LIN {X 0,Y 467.676,Z 280.243,A -85,B 0,C 180,E1 -7671.63,E2 -7671.63} C_VEL
LIN {X 0,Y 467.961,Z 272.023,A -85,B 0,C 180,E1 -7674.393,E2 -7674.393} C_VEL
LIN {X 0,Y 468.313,Z 262.63,A -85,B 0,C 180,E1 -7677.724,E2 -7677.724} C_VEL
LIN {X 0,Y 468.659,Z 254.669,A -85,B 0,C 180,E1 -7680.654,E2 -7680.654} C_VEL
LIN {X 0,Y 469.091,Z 246.823,A -85,B 0,C 180,E1 -7683.665,E2 -7683.665} C_VEL
LIN {X 0,Y 469.381,Z 240.972,A -85,B 0,C 180,E1 -7686.046,E2 -7686.046} C_VEL
LIN {X 0,Y 468.758,Z 236.725,A -85,B 0,C 180,E1 -7687.93,E2 -7687.93} C_VEL
LIN {X 0,Y 467.6,Z 230.243,A -85,B 0,C 180,E1 -7691.113,E2 -7691.113} C_VEL
LIN {X 0,Y 467.556,Z 230.247,A -85,B 0,C 180,E1 -7693.82,E2 -7693.82} C_VEL
LIN {X 0,Y 467.557,Z 230.246,A -85,B 0,C 180,E1 -7696.255,E2 -7696.255} C_VEL
LIN {X 0,Y 467.586,Z 230.243,A -85,B 0,C 180,E1 -7698.721,E2 -7698.721} C_VEL
LIN {X 0,Y 467.577,Z 230.244,A -85,B 0,C 180,E1 -7701.406,E2 -7701.406} C_VEL
LIN {X 0,Y 467.56,Z 230.247,A -85,B 0,C 180,E1 -7704.26,E2 -7704.26} C_VEL
LIN {X 0,Y 467.582,Z 230.244,A -85,B 0,C 180,E1 -7707.32,E2 -7707.32} C_VEL
LIN {X 0,Y 467.57,Z 230.243,A -85,B 0,C 180,E1 -7710.666,E2 -7710.666} C_VEL
LIN {X 0,Y 467.628,Z 230.239,A -85,B 0,C 180,E1 -7713.199,E2 -7713.199} C_VEL
LIN {X 0,Y 467.592,Z 230.242,A -85,B 0,C 180,E1 -7716.467,E2 -7716.467} C_VEL
LIN {X 0,Y 467.623,Z 230.236,A -85,B 0,C 180,E1 -7719.776,E2 -7719.776} C_VEL
LIN {X 0,Y 467.608,Z 230.238,A -85,B 0,C 180,E1 -7722.505,E2 -7722.505} C_VEL
LIN {X 0,Y 467.604,Z 230.24,A -85,B 0,C 180,E1 -7725.195,E2 -7725.195} C_VEL
LIN {X 0,Y 467.653,Z 230.236,A -85,B 0,C 180,E1 -7727.853,E2 -7727.853} C_VEL
LIN {X 0,Y 467.679,Z 230.229,A -85,B 0,C 180,E1 -7731.356,E2 -7731.356} C_VEL
LIN {X 0,Y 467.741,Z 230.222,A -85,B 0,C 180,E1 -7733.961,E2 -7733.961} C_VEL
LIN {X 0,Y 467.857,Z 230.208,A -85,B 0,C 180,E1 -7737.416,E2 -7737.416} C_VEL
LIN {X 0,Y 467.878,Z 230.206,A -85,B 0,C 180,E1 -7739.999,E2 -7739.999} C_VEL
LIN {X 0,Y 467.855,Z 230.209,A -85,B 0,C 180,E1 -7742.581,E2 -7742.581} C_VEL
LIN {X 0,Y 467.738,Z 230.224,A -85,B 0,C 180,E1 -7746.036,E2 -7746.036} C_VEL
LIN {X 0,Y 467.676,Z 230.233,A -85,B 0,C 180,E1 -7748.641,E2 -7748.641} C_VEL
LIN {X 0,Y 467.592,Z 230.245,A -85,B 0,C 180,E1 -7751.266,E2 -7751.266} C_VEL
LIN {X 0,Y 467.277,Z 230.507,A -85,B 0,C 180,E1 -7753.923,E2 -7753.923} C_VEL
LIN {X 0,Y 467.233,Z 233.257,A -85,B 0,C 180,E1 -7756.604,E2 -7756.604} C_VEL
LIN {X 0,Y 467.155,Z 236.019,A -85,B 0,C 180,E1 -7759.326,E2 -7759.326} C_VEL
LIN {X 0,Y 467.074,Z 238.94,A -85,B 0,C 180,E1 -7762.095,E2 -7762.095} C_VEL
LIN {X 0,Y 467.043,Z 241.899,A -85,B 0,C 180,E1 -7764.917,E2 -7764.917} C_VEL
LIN {X 0,Y 466.93,Z 244.936,A -85,B 0,C 180,E1 -7767.812,E2 -7767.812} C_VEL
LIN {X 0,Y 466.869,Z 248.241,A -85,B 0,C 180,E1 -7770.903,E2 -7770.903} C_VEL
LIN {X 0,Y 466.884,Z 249.126,A -85,B 0,C 180,E1 -7771.731,E2 -7771.731} C_VEL
LIN {X 0,Y 470.12,Z 262.455,A -85,B 0,C 180,E1 -7772.256,E2 -7772.256} C_VEL
LIN {X 0,Y 470.316,Z 267.493,A -85,B 0,C 180,E1 -7772.469,E2 -7772.469} C_VEL
LIN {X 0,Y 469.881,Z 280.326,A -85,B 0,C 180,E1 -7773.115,E2 -7773.115} C_VEL
LIN {X 0,Y 469.378,Z 291.965,A -85,B 0,C 180,E1 -7773.898,E2 -7773.898} C_VEL
LIN {X 0,Y 468.916,Z 303.063,A -85,B 0,C 180,E1 -7774.846,E2 -7774.846} C_VEL
LIN {X 0,Y 468.446,Z 312.887,A -85,B 0,C 180,E1 -7775.891,E2 -7775.891} C_VEL
LIN {X 0,Y 468.022,Z 321.872,A -85,B 0,C 180,E1 -7777.077,E2 -7777.077} C_VEL
LIN {X 0,Y 467.606,Z 329.48,A -85,B 0,C 180,E1 -7778.311,E2 -7778.311} C_VEL
LIN {X 0,Y 467.302,Z 335.582,A -85,B 0,C 180,E1 -7779.53,E2 -7779.53} C_VEL
LIN {X 0,Y 467.087,Z 340.512,A -85,B 0,C 180,E1 -7780.753,E2 -7780.753} C_VEL
LIN {X 0,Y 466.944,Z 344.398,A -85,B 0,C 180,E1 -7781.972,E2 -7781.972} C_VEL
LIN {X 0,Y 466.825,Z 347.337,A -85,B 0,C 180,E1 -7783.177,E2 -7783.177} C_VEL
LIN {X 0,Y 466.665,Z 350.158,A -85,B 0,C 180,E1 -7784.943,E2 -7784.943} C_VEL
LIN {X 0,Y 466.633,Z 351.147,A -85,B 0,C 180,E1 -7786.294,E2 -7786.294} C_VEL
LIN {X 0,Y 466.618,Z 351.185,A -85,B 0,C 180,E1 -7787.56,E2 -7787.56} C_VEL
LIN {X 0,Y 466.646,Z 350.357,A -85,B 0,C 180,E1 -7788.851,E2 -7788.851} C_VEL
LIN {X 0,Y 466.745,Z 348.596,A -85,B 0,C 180,E1 -7790.165,E2 -7790.165} C_VEL
LIN {X 0,Y 466.885,Z 344.834,A -85,B 0,C 180,E1 -7791.891,E2 -7791.891} C_VEL
LIN {X 0,Y 467.095,Z 339.496,A -85,B 0,C 180,E1 -7793.536,E2 -7793.536} C_VEL
LIN {X 0,Y 467.374,Z 333.457,A -85,B 0,C 180,E1 -7794.944,E2 -7794.944} C_VEL
LIN {X 0,Y 467.669,Z 326.553,A -85,B 0,C 180,E1 -7796.219,E2 -7796.219} C_VEL
LIN {X 0,Y 468.159,Z 317.583,A -85,B 0,C 180,E1 -7797.543,E2 -7797.543} C_VEL
LIN {X 0,Y 468.545,Z 309,A -85,B 0,C 180,E1 -7798.576,E2 -7798.576} C_VEL
LIN {X 0,Y 469.032,Z 298.415,A -85,B 0,C 180,E1 -7799.614,E2 -7799.614} C_VEL
LIN {X 0,Y 469.515,Z 286.668,A -85,B 0,C 180,E1 -7800.522,E2 -7800.522} C_VEL
LIN {X 0,Y 469.957,Z 274.999,A -85,B 0,C 180,E1 -7801.227,E2 -7801.227} C_VEL
LIN {X 0,Y 470.132,Z 262.702,A -85,B 0,C 180,E1 -7801.787,E2 -7801.787} C_VEL
LIN {X 0,Y 467.551,Z 251.251,A -85,B 0,C 180,E1 -7802.245,E2 -7802.245} C_VEL
LIN {X 0,Y 466.704,Z 249.393,A -85,B 0,C 180,E1 -7802.401,E2 -7802.401} C_VEL
LIN {X 0,Y 465.362,Z 248.01,A -85,B 0,C 180,E1 -7802.739,E2 -7802.739} C_VEL
LIN {X 0,Y 462.544,Z 247.044,A -85,B 0,C 180,E1 -7803.723,E2 -7803.723} C_VEL
LIN {X 0,Y 460.557,Z 246.182,A -85,B 0,C 180,E1 -7804.819,E2 -7804.819} C_VEL
LIN {X 0,Y 459.773,Z 244.848,A -85,B 0,C 180,E1 -7805.933,E2 -7805.933} C_VEL
LIN {X 0,Y 459.817,Z 241.701,A -85,B 0,C 180,E1 -7808.797,E2 -7808.797} C_VEL
LIN {X 0,Y 459.935,Z 238.951,A -85,B 0,C 180,E1 -7811.324,E2 -7811.324} C_VEL
LIN {X 0,Y 459.981,Z 235.075,A -85,B 0,C 180,E1 -7814.946,E2 -7814.946} C_VEL
LIN {X 0,Y 460.104,Z 231.233,A -85,B 0,C 180,E1 -7818.547,E2 -7818.547} C_VEL
LIN {X 0,Y 460.424,Z 231.136,A -85,B 0,C 180,E1 -7821.22,E2 -7821.22} C_VEL
LIN {X 0,Y 460.693,Z 231.1,A -85,B 0,C 180,E1 -7823.87,E2 -7823.87} C_VEL
LIN {X 0,Y 460.81,Z 231.087,A -85,B 0,C 180,E1 -7827.378,E2 -7827.378} C_VEL
LIN {X 0,Y 460.837,Z 231.081,A -85,B 0,C 180,E1 -7830,E2 -7830} C_VEL
LIN {X 0,Y 460.81,Z 231.085,A -85,B 0,C 180,E1 -7832.623,E2 -7832.623} C_VEL
LIN {X 0,Y 460.698,Z 231.098,A -85,B 0,C 180,E1 -7836.131,E2 -7836.131} C_VEL
LIN {X 0,Y 460.614,Z 231.11,A -85,B 0,C 180,E1 -7838.777,E2 -7838.777} C_VEL
LIN {X 0,Y 460.618,Z 231.109,A -85,B 0,C 180,E1 -7842.458,E2 -7842.458} C_VEL
LIN {X 0,Y 460.584,Z 231.113,A -85,B 0,C 180,E1 -7845.999,E2 -7845.999} C_VEL
LIN {X 0,Y 460.556,Z 231.118,A -85,B 0,C 180,E1 -7848.903,E2 -7848.903} C_VEL
LIN {X 0,Y 460.55,Z 231.118,A -85,B 0,C 180,E1 -7851.484,E2 -7851.484} C_VEL
LIN {X 0,Y 460.535,Z 231.119,A -85,B 0,C 180,E1 -7854.333,E2 -7854.333} C_VEL
LIN {X 0,Y 460.57,Z 231.115,A -85,B 0,C 180,E1 -7857.244,E2 -7857.244} C_VEL
LIN {X 0,Y 460.498,Z 231.124,A -85,B 0,C 180,E1 -7860.241,E2 -7860.241} C_VEL
LIN {X 0,Y 460.517,Z 231.121,A -85,B 0,C 180,E1 -7863.326,E2 -7863.326} C_VEL
LIN {X 0,Y 460.468,Z 231.13,A -85,B 0,C 180,E1 -7866.531,E2 -7866.531} C_VEL
LIN {X 0,Y 460.568,Z 231.115,A -85,B 0,C 180,E1 -7869.859,E2 -7869.859} C_VEL
LIN {X 0,Y 460.532,Z 231.12,A -85,B 0,C 180,E1 -7872.906,E2 -7872.906} C_VEL
LIN {X 0,Y 460.515,Z 231.122,A -85,B 0,C 180,E1 -7875.83,E2 -7875.83} C_VEL
LIN {X 0,Y 460.535,Z 231.12,A -85,B 0,C 180,E1 -7878.992,E2 -7878.992} C_VEL
LIN {X 0,Y 460.539,Z 231.118,A -85,B 0,C 180,E1 -7881.271,E2 -7881.271} C_VEL
LIN {X 0,Y 460.506,Z 231.124,A -85,B 0,C 180,E1 -7884.556,E2 -7884.556} C_VEL
LIN {X 0,Y 460.527,Z 231.12,A -85,B 0,C 180,E1 -7887.718,E2 -7887.718} C_VEL
LIN {X 0,Y 460.543,Z 231.119,A -85,B 0,C 180,E1 -7890.771,E2 -7890.771} C_VEL
LIN {X 0,Y 460.559,Z 231.117,A -85,B 0,C 180,E1 -7893.737,E2 -7893.737} C_VEL
LIN {X 0,Y 460.543,Z 231.119,A -85,B 0,C 180,E1 -7896.626,E2 -7896.626} C_VEL
LIN {X 0,Y 460.549,Z 231.117,A -85,B 0,C 180,E1 -7899.455,E2 -7899.455} C_VEL
LIN {X 0,Y 460.559,Z 231.118,A -85,B 0,C 180,E1 -7902.232,E2 -7902.232} C_VEL
LIN {X 0,Y 460.564,Z 231.114,A -85,B 0,C 180,E1 -7904.967,E2 -7904.967} C_VEL
LIN {X 0,Y 460.61,Z 231.11,A -85,B 0,C 180,E1 -7908.561,E2 -7908.561} C_VEL
LIN {X 0,Y 460.619,Z 231.108,A -85,B 0,C 180,E1 -7911.225,E2 -7911.225} C_VEL
LIN {X 0,Y 460.708,Z 231.1,A -85,B 0,C 180,E1 -7913.872,E2 -7913.872} C_VEL
LIN {X 0,Y 460.801,Z 231.087,A -85,B 0,C 180,E1 -7917.379,E2 -7917.379} C_VEL
LIN {X 0,Y 460.855,Z 231.082,A -85,B 0,C 180,E1 -7920.001,E2 -7920.001} C_VEL
LIN {X 0,Y 460.801,Z 231.086,A -85,B 0,C 180,E1 -7922.624,E2 -7922.624} C_VEL
LIN {X 0,Y 460.689,Z 231.1,A -85,B 0,C 180,E1 -7926.132,E2 -7926.132} C_VEL
LIN {X 0,Y 460.623,Z 231.108,A -85,B 0,C 180,E1 -7928.778,E2 -7928.778} C_VEL
LIN {X 0,Y 460.618,Z 231.107,A -85,B 0,C 180,E1 -7932.446,E2 -7932.446} C_VEL
LIN {X 0,Y 460.605,Z 231.111,A -85,B 0,C 180,E1 -7935.999,E2 -7935.999} C_VEL
LIN {X 0,Y 460.576,Z 231.114,A -85,B 0,C 180,E1 -7938.903,E2 -7938.903} C_VEL
LIN {X 0,Y 460.521,Z 231.124,A -85,B 0,C 180,E1 -7941.487,E2 -7941.487} C_VEL
LIN {X 0,Y 460.527,Z 231.119,A -85,B 0,C 180,E1 -7944.334,E2 -7944.334} C_VEL
LIN {X 0,Y 460.564,Z 231.118,A -85,B 0,C 180,E1 -7947.246,E2 -7947.246} C_VEL
LIN {X 0,Y 460.516,Z 231.121,A -85,B 0,C 180,E1 -7950.241,E2 -7950.241} C_VEL
LIN {X 0,Y 460.526,Z 231.124,A -85,B 0,C 180,E1 -7953.326,E2 -7953.326} C_VEL
LIN {X 0,Y 460.482,Z 231.125,A -85,B 0,C 180,E1 -7956.53,E2 -7956.53} C_VEL
LIN {X 0,Y 460.533,Z 231.119,A -85,B 0,C 180,E1 -7959.863,E2 -7959.863} C_VEL
LIN {X 0,Y 460.518,Z 231.121,A -85,B 0,C 180,E1 -7962.901,E2 -7962.901} C_VEL
LIN {X 0,Y 460.513,Z 231.121,A -85,B 0,C 180,E1 -7965.831,E2 -7965.831} C_VEL
LIN {X 0,Y 460.572,Z 231.225,A -85,B 0,C 180,E1 -7968.772,E2 -7968.772} C_VEL
LIN {X 0,Y 461.795,Z 237.98,A -85,B 0,C 180,E1 -7971.885,E2 -7971.885} C_VEL
LIN {X 0,Y 462.378,Z 242.064,A -85,B 0,C 180,E1 -7973.668,E2 -7973.668} C_VEL
LIN {X 0,Y 462.268,Z 247.187,A -85,B 0,C 180,E1 -7975.769,E2 -7975.769} C_VEL
LIN {X 0,Y 461.823,Z 255.013,A -85,B 0,C 180,E1 -7978.841,E2 -7978.841} C_VEL
LIN {X 0,Y 461.394,Z 263.555,A -85,B 0,C 180,E1 -7982.064,E2 -7982.064} C_VEL
LIN {X 0,Y 460.978,Z 272.095,A -85,B 0,C 180,E1 -7985.212,E2 -7985.212} C_VEL
LIN {X 0,Y 460.666,Z 281.728,A -85,B 0,C 180,E1 -7988.534,E2 -7988.534} C_VEL
LIN {X 0,Y 460.372,Z 291.269,A -85,B 0,C 180,E1 -7991.762,E2 -7991.762} C_VEL
LIN {X 0,Y 460.171,Z 299.065,A -85,B 0,C 180,E1 -7994.352,E2 -7994.352} C_VEL
LIN {X 0,Y 462.488,Z 312.664,A -85,B 0,C 180,E1 -7994.786,E2 -7994.786} C_VEL
LIN {X 0,Y 463.263,Z 319.162,A -85,B 0,C 180,E1 -7995.054,E2 -7995.054} C_VEL
LIN {X 0,Y 462.85,Z 330.828,A -85,B 0,C 180,E1 -7995.602,E2 -7995.602} C_VEL
LIN {X 0,Y 462.346,Z 341.575,A -85,B 0,C 180,E1 -7996.26,E2 -7996.26} C_VEL
LIN {X 0,Y 461.85,Z 353.16,A -85,B 0,C 180,E1 -7997.161,E2 -7997.161} C_VEL
LIN {X 0,Y 461.377,Z 363.168,A -85,B 0,C 180,E1 -7998.133,E2 -7998.133} C_VEL
LIN {X 0,Y 460.819,Z 372.383,A -85,B 0,C 180,E1 -7999.232,E2 -7999.232} C_VEL
LIN {X 0,Y 460.42,Z 381.376,A -85,B 0,C 180,E1 -8000.555,E2 -8000.555} C_VEL
LIN {X 0,Y 460.057,Z 388.614,A -85,B 0,C 180,E1 -8001.876,E2 -8001.876} C_VEL
LIN {X 0,Y 459.851,Z 393.504,A -85,B 0,C 180,E1 -8002.977,E2 -8002.977} C_VEL
LIN {X 0,Y 459.755,Z 398.263,A -85,B 0,C 180,E1 -8004.297,E2 -8004.297} C_VEL
LIN {X 0,Y 459.581,Z 401.894,A -85,B 0,C 180,E1 -8005.614,E2 -8005.614} C_VEL
LIN {X 0,Y 459.592,Z 403.772,A -85,B 0,C 180,E1 -8006.493,E2 -8006.493} C_VEL
LIN {X 0,Y 459.572,Z 405.175,A -85,B 0,C 180,E1 -8007.37,E2 -8007.37} C_VEL
LIN {X 0,Y 459.496,Z 406.778,A -85,B 0,C 180,E1 -8009.123,E2 -8009.123} C_VEL
LIN {X 0,Y 459.475,Z 406.994,A -85,B 0,C 180,E1 -8010,E2 -8010} C_VEL
LIN {X 0,Y 459.496,Z 406.779,A -85,B 0,C 180,E1 -8010.876,E2 -8010.876} C_VEL
LIN {X 0,Y 459.572,Z 405.179,A -85,B 0,C 180,E1 -8012.629,E2 -8012.629} C_VEL
LIN {X 0,Y 459.592,Z 403.778,A -85,B 0,C 180,E1 -8013.506,E2 -8013.506} C_VEL
LIN {X 0,Y 459.635,Z 400.819,A -85,B 0,C 180,E1 -8014.824,E2 -8014.824} C_VEL
LIN {X 0,Y 459.759,Z 396.815,A -85,B 0,C 180,E1 -8016.142,E2 -8016.142} C_VEL
LIN {X 0,Y 459.928,Z 390.656,A -85,B 0,C 180,E1 -8017.683,E2 -8017.683} C_VEL
LIN {X 0,Y 460.288,Z 383.936,A -85,B 0,C 180,E1 -8019.003,E2 -8019.003} C_VEL
LIN {X 0,Y 460.701,Z 375.598,A -85,B 0,C 180,E1 -8020.325,E2 -8020.325} C_VEL
LIN {X 0,Y 461.152,Z 367.056,A -85,B 0,C 180,E1 -8021.427,E2 -8021.427} C_VEL
LIN {X 0,Y 461.674,Z 356.888,A -85,B 0,C 180,E1 -8022.492,E2 -8022.492} C_VEL
LIN {X 0,Y 462.091,Z 346.077,A -85,B 0,C 180,E1 -8023.411,E2 -8023.411} C_VEL
LIN {X 0,Y 462.652,Z 334.667,A -85,B 0,C 180,E1 -8024.178,E2 -8024.178} C_VEL
LIN {X 0,Y 463.12,Z 322.971,A -85,B 0,C 180,E1 -8024.781,E2 -8024.781} C_VEL
LIN {X 0,Y 462.988,Z 316.237,A -85,B 0,C 180,E1 -8025.063,E2 -8025.063} C_VEL
LIN {X 0,Y 460.789,Z 302.835,A -85,B 0,C 180,E1 -8025.543,E2 -8025.543} C_VEL
LIN {X 0,Y 460.148,Z 298.602,A -85,B 0,C 180,E1 -8025.688,E2 -8025.688} C_VEL
LIN {X 0,Y 460.454,Z 288.214,A -85,B 0,C 180,E1 -8029.178,E2 -8029.178} C_VEL
LIN {X 0,Y 460.706,Z 278.58,A -85,B 0,C 180,E1 -8032.418,E2 -8032.418} C_VEL
LIN {X 0,Y 460.982,Z 270.434,A -85,B 0,C 180,E1 -8035.269,E2 -8035.269} C_VEL
LIN {X 0,Y 461.352,Z 262.326,A -85,B 0,C 180,E1 -8038.179,E2 -8038.179} C_VEL
LIN {X 0,Y 461.747,Z 253.505,A -85,B 0,C 180,E1 -8041.531,E2 -8041.531} C_VEL
LIN {X 0,Y 462.294,Z 245.24,A -85,B 0,C 180,E1 -8044.821,E2 -8044.821} C_VEL
LIN {X 0,Y 462.338,Z 241.624,A -85,B 0,C 180,E1 -8046.358,E2 -8046.358} C_VEL
LIN {X 0,Y 461.367,Z 235.858,A -85,B 0,C 180,E1 -8049.023,E2 -8049.023} C_VEL
LIN {X 0,Y 460.527,Z 231.125,A -85,B 0,C 180,E1 -8051.492,E2 -8051.492} C_VEL
LIN {X 0,Y 460.518,Z 231.124,A -85,B 0,C 180,E1 -8054.587,E2 -8054.587} C_VEL
LIN {X 0,Y 460.525,Z 231.123,A -85,B 0,C 180,E1 -8057.818,E2 -8057.818} C_VEL
LIN {X 0,Y 460.568,Z 231.118,A -85,B 0,C 180,E1 -8061.098,E2 -8061.098} C_VEL
LIN {X 0,Y 460.51,Z 231.125,A -85,B 0,C 180,E1 -8064.553,E2 -8064.553} C_VEL
LIN {X 0,Y 460.531,Z 231.122,A -85,B 0,C 180,E1 -8067.714,E2 -8067.714} C_VEL
LIN {X 0,Y 460.54,Z 231.119,A -85,B 0,C 180,E1 -8070.768,E2 -8070.768} C_VEL
LIN {X 0,Y 460.568,Z 231.116,A -85,B 0,C 180,E1 -8073.734,E2 -8073.734} C_VEL
LIN {X 0,Y 460.545,Z 231.119,A -85,B 0,C 180,E1 -8076.623,E2 -8076.623} C_VEL
LIN {X 0,Y 460.551,Z 231.118,A -85,B 0,C 180,E1 -8079.452,E2 -8079.452} C_VEL
LIN {X 0,Y 460.558,Z 231.115,A -85,B 0,C 180,E1 -8082.229,E2 -8082.229} C_VEL
LIN {X 0,Y 460.563,Z 231.117,A -85,B 0,C 180,E1 -8084.964,E2 -8084.964} C_VEL
LIN {X 0,Y 460.608,Z 231.112,A -85,B 0,C 180,E1 -8088.558,E2 -8088.558} C_VEL
LIN {X 0,Y 460.692,Z 231.102,A -85,B 0,C 180,E1 -8092.107,E2 -8092.107} C_VEL
LIN {X 0,Y 460.695,Z 231.101,A -85,B 0,C 180,E1 -8094.747,E2 -8094.747} C_VEL
LIN {X 0,Y 460.822,Z 231.084,A -85,B 0,C 180,E1 -8097.376,E2 -8097.376} C_VEL
LIN {X 0,Y 460.849,Z 231.081,A -85,B 0,C 180,E1 -8099.999,E2 -8099.999} C_VEL
LIN {X 0,Y 460.82,Z 231.085,A -85,B 0,C 180,E1 -8102.621,E2 -8102.621} C_VEL
LIN {X 0,Y 460.704,Z 231.101,A -85,B 0,C 180,E1 -8106.128,E2 -8106.128} C_VEL
LIN {X 0,Y 460.622,Z 231.111,A -85,B 0,C 180,E1 -8108.775,E2 -8108.775} C_VEL
LIN {X 0,Y 460.541,Z 231.124,A -85,B 0,C 180,E1 -8111.441,E2 -8111.441} C_VEL
LIN {X 0,Y 460.311,Z 231.153,A -85,B 0,C 180,E1 -8113.238,E2 -8113.238} C_VEL
LIN {X 0,Y 460.242,Z 231.62,A -85,B 0,C 180,E1 -8114.14,E2 -8114.14} C_VEL
LIN {X 0,Y 460.168,Z 234.362,A -85,B 0,C 180,E1 -8116.867,E2 -8116.867} C_VEL
LIN {X 0,Y 460.079,Z 237.194,A -85,B 0,C 180,E1 -8119.635,E2 -8119.635} C_VEL
LIN {X 0,Y 460.027,Z 240.113,A -85,B 0,C 180,E1 -8122.452,E2 -8122.452} C_VEL
LIN {X 0,Y 459.947,Z 243.418,A -85,B 0,C 180,E1 -8125.643,E2 -8125.643} C_VEL
LIN {X 0,Y 459.877,Z 246.184,A -85,B 0,C 180,E1 -8128.276,E2 -8128.276} C_VEL
LIN {X 0,Y 459.818,Z 249.552,A -85,B 0,C 180,E1 -8131.468,E2 -8131.468} C_VEL
LIN {X 0,Y 463.413,Z 264.288,A -85,B 0,C 180,E1 -8132.089,E2 -8132.089} C_VEL
LIN {X 0,Y 463.201,Z 276.299,A -85,B 0,C 180,E1 -8132.653,E2 -8132.653} C_VEL
LIN {X 0,Y 462.697,Z 287.558,A -85,B 0,C 180,E1 -8133.343,E2 -8133.343} C_VEL
LIN {X 0,Y 462.225,Z 298.872,A -85,B 0,C 180,E1 -8134.232,E2 -8134.232} C_VEL
LIN {X 0,Y 461.748,Z 308.535,A -85,B 0,C 180,E1 -8135.174,E2 -8135.174} C_VEL
LIN {X 0,Y 461.254,Z 317.661,A -85,B 0,C 180,E1 -8136.268,E2 -8136.268} C_VEL
LIN {X 0,Y 460.768,Z 326.595,A -85,B 0,C 180,E1 -8137.595,E2 -8137.595} C_VEL
LIN {X 0,Y 460.409,Z 333.548,A -85,B 0,C 180,E1 -8138.878,E2 -8138.878} C_VEL
LIN {X 0,Y 460.097,Z 339.319,A -85,B 0,C 180,E1 -8140.205,E2 -8140.205} C_VEL
LIN {X 0,Y 459.921,Z 343.793,A -85,B 0,C 180,E1 -8141.518,E2 -8141.518} C_VEL
LIN {X 0,Y 459.815,Z 347.138,A -85,B 0,C 180,E1 -8142.808,E2 -8142.808} C_VEL
LIN {X 0,Y 459.669,Z 349.474,A -85,B 0,C 180,E1 -8144.062,E2 -8144.062} C_VEL
LIN {X 0,Y 459.572,Z 350.948,A -85,B 0,C 180,E1 -8145.296,E2 -8145.296} C_VEL
LIN {X 0,Y 459.545,Z 351.64,A -85,B 0,C 180,E1 -8146.513,E2 -8146.513} C_VEL
LIN {X 0,Y 459.528,Z 351.586,A -85,B 0,C 180,E1 -8147.707,E2 -8147.707} C_VEL
LIN {X 0,Y 459.561,Z 350.776,A -85,B 0,C 180,E1 -8148.884,E2 -8148.884} C_VEL
LIN {X 0,Y 459.659,Z 349.29,A -85,B 0,C 180,E1 -8150.048,E2 -8150.048} C_VEL
LIN {X 0,Y 459.823,Z 345.737,A -85,B 0,C 180,E1 -8151.771,E2 -8151.771} C_VEL
LIN {X 0,Y 459.957,Z 342.06,A -85,B 0,C 180,E1 -8153.023,E2 -8153.023} C_VEL
LIN {X 0,Y 460.222,Z 336.297,A -85,B 0,C 180,E1 -8154.53,E2 -8154.53} C_VEL
LIN {X 0,Y 460.535,Z 329.598,A -85,B 0,C 180,E1 -8155.888,E2 -8155.888} C_VEL
LIN {X 0,Y 460.974,Z 321.226,A -85,B 0,C 180,E1 -8157.247,E2 -8157.247} C_VEL
LIN {X 0,Y 461.467,Z 312.508,A -85,B 0,C 180,E1 -8158.391,E2 -8158.391} C_VEL
LIN {X 0,Y 461.926,Z 302.199,A -85,B 0,C 180,E1 -8159.484,E2 -8159.484} C_VEL
LIN {X 0,Y 462.476,Z 291.384,A -85,B 0,C 180,E1 -8160.404,E2 -8160.404} C_VEL
LIN {X 0,Y 462.888,Z 279.931,A -85,B 0,C 180,E1 -8161.181,E2 -8161.181} C_VEL
LIN {X 0,Y 463.322,Z 267.962,A -85,B 0,C 180,E1 -8161.794,E2 -8161.794} C_VEL
LIN {X 0,Y 463.355,Z 264.283,A -85,B 0,C 180,E1 -8161.954,E2 -8161.954} C_VEL
LIN {X 0,Y 460.442,Z 251.546,A -85,B 0,C 180,E1 -8162.48,E2 -8162.48} C_VEL
LIN {X 0,Y 459.802,Z 248.539,A -85,B 0,C 180,E1 -8162.61,E2 -8162.61} C_VEL
LIN {X 0,Y 459.781,Z 245.192,A -85,B 0,C 180,E1 -8165.626,E2 -8165.626} C_VEL
LIN {X 0,Y 459.773,Z 244.848,A -85,B 0,C 180,E1 -8165.933,E2 -8165.933} C_VEL
LIN {X 0,Y 459.109,Z 244.106,A -85,B 0,C 180,E1 -8166.659,E2 -8166.659} C_VEL
LIN {X 0,Y 456.253,Z 243.084,A -85,B 0,C 180,E1 -8167.841,E2 -8167.841} C_VEL
LIN {X 0,Y 453.843,Z 242.295,A -85,B 0,C 180,E1 -8168.795,E2 -8168.795} C_VEL
LIN {X 0,Y 452.819,Z 241.589,A -85,B 0,C 180,E1 -8169.531,E2 -8169.531} C_VEL
LIN {X 0,Y 452.742,Z 241.324,A -85,B 0,C 180,E1 -8169.779,E2 -8169.779} C_VEL
LIN {X 0,Y 452.847,Z 239.011,A -85,B 0,C 180,E1 -8171.918,E2 -8171.918} C_VEL
LIN {X 0,Y 452.911,Z 236.037,A -85,B 0,C 180,E1 -8174.705,E2 -8174.705} C_VEL
LIN {X 0,Y 453.03,Z 232.177,A -85,B 0,C 180,E1 -8178.366,E2 -8178.366} C_VEL
LIN {X 0,Y 453.37,Z 232.014,A -85,B 0,C 180,E1 -8181.083,E2 -8181.083} C_VEL
LIN {X 0,Y 453.657,Z 231.977,A -85,B 0,C 180,E1 -8183.775,E2 -8183.775} C_VEL
LIN {X 0,Y 453.75,Z 231.966,A -85,B 0,C 180,E1 -8187.337,E2 -8187.337} C_VEL
LIN {X 0,Y 453.807,Z 231.957,A -85,B 0,C 180,E1 -8190,E2 -8190} C_VEL
LIN {X 0,Y 453.751,Z 231.964,A -85,B 0,C 180,E1 -8192.664,E2 -8192.664} C_VEL
LIN {X 0,Y 453.665,Z 231.974,A -85,B 0,C 180,E1 -8196.226,E2 -8196.226} C_VEL
LIN {X 0,Y 453.578,Z 231.988,A -85,B 0,C 180,E1 -8198.914,E2 -8198.914} C_VEL
LIN {X 0,Y 453.586,Z 231.986,A -85,B 0,C 180,E1 -8202.552,E2 -8202.552} C_VEL
LIN {X 0,Y 453.529,Z 231.992,A -85,B 0,C 180,E1 -8206.197,E2 -8206.197} C_VEL
LIN {X 0,Y 453.506,Z 231.996,A -85,B 0,C 180,E1 -8209.042,E2 -8209.042} C_VEL
LIN {X 0,Y 453.489,Z 231.997,A -85,B 0,C 180,E1 -8211.836,E2 -8211.836} C_VEL
LIN {X 0,Y 453.513,Z 231.996,A -85,B 0,C 180,E1 -8214.735,E2 -8214.735} C_VEL
LIN {X 0,Y 453.524,Z 231.992,A -85,B 0,C 180,E1 -8217.962,E2 -8217.962} C_VEL
LIN {X 0,Y 453.454,Z 232.001,A -85,B 0,C 180,E1 -8221.527,E2 -8221.527} C_VEL
LIN {X 0,Y 453.477,Z 232,A -85,B 0,C 180,E1 -8224.779,E2 -8224.779} C_VEL
LIN {X 0,Y 453.474,Z 232,A -85,B 0,C 180,E1 -8228.311,E2 -8228.311} C_VEL
LIN {X 0,Y 453.506,Z 231.996,A -85,B 0,C 180,E1 -8230.608,E2 -8230.608} C_VEL
LIN {X 0,Y 453.472,Z 232,A -85,B 0,C 180,E1 -8233.249,E2 -8233.249} C_VEL
LIN {X 0,Y 453.468,Z 231.999,A -85,B 0,C 180,E1 -8235.782,E2 -8235.782} C_VEL
LIN {X 0,Y 453.488,Z 231.999,A -85,B 0,C 180,E1 -8238.213,E2 -8238.213} C_VEL
LIN {X 0,Y 453.525,Z 231.993,A -85,B 0,C 180,E1 -8240.789,E2 -8240.789} C_VEL
LIN {X 0,Y 453.45,Z 232.002,A -85,B 0,C 180,E1 -8243.919,E2 -8243.919} C_VEL
LIN {X 0,Y 453.477,Z 231.997,A -85,B 0,C 180,E1 -8247.153,E2 -8247.153} C_VEL
LIN {X 0,Y 453.509,Z 231.997,A -85,B 0,C 180,E1 -8250.273,E2 -8250.273} C_VEL
LIN {X 0,Y 453.505,Z 231.993,A -85,B 0,C 180,E1 -8253.296,E2 -8253.296} C_VEL
LIN {X 0,Y 453.501,Z 231.998,A -85,B 0,C 180,E1 -8256.241,E2 -8256.241} C_VEL
LIN {X 0,Y 453.48,Z 231.996,A -85,B 0,C 180,E1 -8259.119,E2 -8259.119} C_VEL
LIN {X 0,Y 453.511,Z 231.996,A -85,B 0,C 180,E1 -8261.946,E2 -8261.946} C_VEL
LIN {X 0,Y 453.539,Z 231.99,A -85,B 0,C 180,E1 -8264.728,E2 -8264.728} C_VEL
LIN {X 0,Y 453.559,Z 231.989,A -85,B 0,C 180,E1 -8268.381,E2 -8268.381} C_VEL
LIN {X 0,Y 453.585,Z 231.984,A -85,B 0,C 180,E1 -8271.088,E2 -8271.088} C_VEL
LIN {X 0,Y 453.674,Z 231.976,A -85,B 0,C 180,E1 -8273.776,E2 -8273.776} C_VEL
LIN {X 0,Y 453.745,Z 231.965,A -85,B 0,C 180,E1 -8277.338,E2 -8277.338} C_VEL
LIN {X 0,Y 453.825,Z 231.957,A -85,B 0,C 180,E1 -8280.001,E2 -8280.001} C_VEL
LIN {X 0,Y 453.745,Z 231.964,A -85,B 0,C 180,E1 -8282.665,E2 -8282.665} C_VEL
LIN {X 0,Y 453.654,Z 231.976,A -85,B 0,C 180,E1 -8286.227,E2 -8286.227} C_VEL
LIN {X 0,Y 453.589,Z 231.985,A -85,B 0,C 180,E1 -8288.915,E2 -8288.915} C_VEL
LIN {X 0,Y 453.568,Z 231.985,A -85,B 0,C 180,E1 -8292.53,E2 -8292.53} C_VEL
LIN {X 0,Y 453.55,Z 231.99,A -85,B 0,C 180,E1 -8296.197,E2 -8296.197} C_VEL
LIN {X 0,Y 453.526,Z 231.993,A -85,B 0,C 180,E1 -8299.042,E2 -8299.042} C_VEL
LIN {X 0,Y 453.482,Z 231.998,A -85,B 0,C 180,E1 -8301.837,E2 -8301.837} C_VEL
LIN {X 0,Y 453.498,Z 231.995,A -85,B 0,C 180,E1 -8304.737,E2 -8304.737} C_VEL
LIN {X 0,Y 453.535,Z 231.991,A -85,B 0,C 180,E1 -8307.96,E2 -8307.96} C_VEL
LIN {X 0,Y 453.471,Z 232,A -85,B 0,C 180,E1 -8311.526,E2 -8311.526} C_VEL
LIN {X 0,Y 453.488,Z 231.999,A -85,B 0,C 180,E1 -8314.777,E2 -8314.777} C_VEL
LIN {X 0,Y 453.469,Z 232.001,A -85,B 0,C 180,E1 -8318.312,E2 -8318.312} C_VEL
LIN {X 0,Y 453.5,Z 231.997,A -85,B 0,C 180,E1 -8320.609,E2 -8320.609} C_VEL
LIN {X 0,Y 453.459,Z 231.999,A -85,B 0,C 180,E1 -8323.244,E2 -8323.244} C_VEL
LIN {X 0,Y 453.468,Z 231.999,A -85,B 0,C 180,E1 -8325.779,E2 -8325.779} C_VEL
LIN {X 0,Y 453.525,Z 232.071,A -85,B 0,C 180,E1 -8328.437,E2 -8328.437} C_VEL
LIN {X 0,Y 454.596,Z 238.029,A -85,B 0,C 180,E1 -8331.242,E2 -8331.242} C_VEL
LIN {X 0,Y 455.337,Z 242.776,A -85,B 0,C 180,E1 -8333.381,E2 -8333.381} C_VEL
LIN {X 0,Y 455.33,Z 247.046,A -85,B 0,C 180,E1 -8335.173,E2 -8335.173} C_VEL
LIN {X 0,Y 454.885,Z 254.841,A -85,B 0,C 180,E1 -8338.311,E2 -8338.311} C_VEL
LIN {X 0,Y 454.392,Z 264.006,A -85,B 0,C 180,E1 -8341.839,E2 -8341.839} C_VEL
LIN {X 0,Y 453.981,Z 271.918,A -85,B 0,C 180,E1 -8344.803,E2 -8344.803} C_VEL
LIN {X 0,Y 453.62,Z 281.413,A -85,B 0,C 180,E1 -8348.171,E2 -8348.171} C_VEL
LIN {X 0,Y 453.323,Z 291.018,A -85,B 0,C 180,E1 -8351.475,E2 -8351.475} C_VEL
LIN {X 0,Y 453.084,Z 298.522,A -85,B 0,C 180,E1 -8354.096,E2 -8354.096} C_VEL
LIN {X 0,Y 455.258,Z 311.582,A -85,B 0,C 180,E1 -8354.517,E2 -8354.517} C_VEL
LIN {X 0,Y 456.343,Z 320.057,A -85,B 0,C 180,E1 -8354.879,E2 -8354.879} C_VEL
LIN {X 0,Y 455.836,Z 332.399,A -85,B 0,C 180,E1 -8355.49,E2 -8355.49} C_VEL
LIN {X 0,Y 455.292,Z 344.288,A -85,B 0,C 180,E1 -8356.27,E2 -8356.27} C_VEL
LIN {X 0,Y 454.78,Z 354.827,A -85,B 0,C 180,E1 -8357.152,E2 -8357.152} C_VEL
LIN {X 0,Y 454.279,Z 364.713,A -85,B 0,C 180,E1 -8358.171,E2 -8358.171} C_VEL
LIN {X 0,Y 453.701,Z 373.602,A -85,B 0,C 180,E1 -8359.287,E2 -8359.287} C_VEL
LIN {X 0,Y 453.312,Z 382.287,A -85,B 0,C 180,E1 -8360.631,E2 -8360.631} C_VEL
LIN {X 0,Y 452.927,Z 389.226,A -85,B 0,C 180,E1 -8361.972,E2 -8361.972} C_VEL
LIN {X 0,Y 452.734,Z 395.368,A -85,B 0,C 180,E1 -8363.47,E2 -8363.47} C_VEL
LIN {X 0,Y 452.568,Z 400.4,A -85,B 0,C 180,E1 -8365.1,E2 -8365.1} C_VEL
LIN {X 0,Y 452.494,Z 403.354,A -85,B 0,C 180,E1 -8366.438,E2 -8366.438} C_VEL
LIN {X 0,Y 452.497,Z 404.763,A -85,B 0,C 180,E1 -8367.329,E2 -8367.329} C_VEL
LIN {X 0,Y 452.434,Z 406.378,A -85,B 0,C 180,E1 -8369.109,E2 -8369.109} C_VEL
LIN {X 0,Y 452.412,Z 406.593,A -85,B 0,C 180,E1 -8370,E2 -8370} C_VEL
LIN {X 0,Y 452.434,Z 406.375,A -85,B 0,C 180,E1 -8370.89,E2 -8370.89} C_VEL
LIN {X 0,Y 452.497,Z 404.759,A -85,B 0,C 180,E1 -8372.67,E2 -8372.67} C_VEL
LIN {X 0,Y 452.495,Z 403.347,A -85,B 0,C 180,E1 -8373.561,E2 -8373.561} C_VEL
LIN {X 0,Y 452.568,Z 400.384,A -85,B 0,C 180,E1 -8374.899,E2 -8374.899} C_VEL
LIN {X 0,Y 452.694,Z 395.499,A -85,B 0,C 180,E1 -8376.485,E2 -8376.485} C_VEL
LIN {X 0,Y 452.926,Z 389.189,A -85,B 0,C 180,E1 -8378.027,E2 -8378.027} C_VEL
LIN {X 0,Y 453.301,Z 382.233,A -85,B 0,C 180,E1 -8379.368,E2 -8379.368} C_VEL
LIN {X 0,Y 453.7,Z 373.531,A -85,B 0,C 180,E1 -8380.712,E2 -8380.712} C_VEL
LIN {X 0,Y 454.275,Z 364.625,A -85,B 0,C 180,E1 -8381.828,E2 -8381.828} C_VEL
LIN {X 0,Y 454.789,Z 354.807,A -85,B 0,C 180,E1 -8382.839,E2 -8382.839} C_VEL
LIN {X 0,Y 455.236,Z 344.165,A -85,B 0,C 180,E1 -8383.73,E2 -8383.73} C_VEL
LIN {X 0,Y 455.852,Z 332.252,A -85,B 0,C 180,E1 -8384.508,E2 -8384.508} C_VEL
LIN {X 0,Y 456.338,Z 319.884,A -85,B 0,C 180,E1 -8385.12,E2 -8385.12} C_VEL
LIN {X 0,Y 454.583,Z 307.448,A -85,B 0,C 180,E1 -8385.629,E2 -8385.629} C_VEL
LIN {X 0,Y 453.105,Z 298.157,A -85,B 0,C 180,E1 -8385.931,E2 -8385.931} C_VEL
LIN {X 0,Y 453.41,Z 287.845,A -85,B 0,C 180,E1 -8389.466,E2 -8389.466} C_VEL
LIN {X 0,Y 453.681,Z 278.219,A -85,B 0,C 180,E1 -8392.784,E2 -8392.784} C_VEL
LIN {X 0,Y 454.032,Z 268.849,A -85,B 0,C 180,E1 -8396.13,E2 -8396.13} C_VEL
LIN {X 0,Y 454.409,Z 260.771,A -85,B 0,C 180,E1 -8399.155,E2 -8399.155} C_VEL
LIN {X 0,Y 454.877,Z 252.943,A -85,B 0,C 180,E1 -8402.211,E2 -8402.211} C_VEL
LIN {X 0,Y 455.385,Z 245.839,A -85,B 0,C 180,E1 -8405.118,E2 -8405.118} C_VEL
LIN {X 0,Y 455.235,Z 241.538,A -85,B 0,C 180,E1 -8407.019,E2 -8407.019} C_VEL
LIN {X 0,Y 453.881,Z 234.101,A -85,B 0,C 180,E1 -8410.647,E2 -8410.647} C_VEL
LIN {X 0,Y 453.481,Z 232.003,A -85,B 0,C 180,E1 -8411.79,E2 -8411.79} C_VEL
LIN {X 0,Y 453.488,Z 232,A -85,B 0,C 180,E1 -8415.47,E2 -8415.47} C_VEL
LIN {X 0,Y 453.483,Z 232,A -85,B 0,C 180,E1 -8418.208,E2 -8418.208} C_VEL
LIN {X 0,Y 453.533,Z 231.995,A -85,B 0,C 180,E1 -8420.786,E2 -8420.786} C_VEL
LIN {X 0,Y 453.454,Z 232.005,A -85,B 0,C 180,E1 -8423.916,E2 -8423.916} C_VEL
LIN {X 0,Y 453.483,Z 232,A -85,B 0,C 180,E1 -8427.15,E2 -8427.15} C_VEL
LIN {X 0,Y 453.475,Z 232,A -85,B 0,C 180,E1 -8430.267,E2 -8430.267} C_VEL
LIN {X 0,Y 453.514,Z 231.996,A -85,B 0,C 180,E1 -8433.293,E2 -8433.293} C_VEL
LIN {X 0,Y 453.503,Z 231.997,A -85,B 0,C 180,E1 -8436.238,E2 -8436.238} C_VEL
LIN {X 0,Y 453.482,Z 231.999,A -85,B 0,C 180,E1 -8439.116,E2 -8439.116} C_VEL
LIN {X 0,Y 453.51,Z 231.993,A -85,B 0,C 180,E1 -8441.943,E2 -8441.943} C_VEL
LIN {X 0,Y 453.538,Z 231.991,A -85,B 0,C 180,E1 -8444.725,E2 -8444.725} C_VEL
LIN {X 0,Y 453.557,Z 231.99,A -85,B 0,C 180,E1 -8448.378,E2 -8448.378} C_VEL
LIN {X 0,Y 453.649,Z 231.978,A -85,B 0,C 180,E1 -8451.984,E2 -8451.984} C_VEL
LIN {X 0,Y 453.669,Z 231.976,A -85,B 0,C 180,E1 -8454.665,E2 -8454.665} C_VEL
LIN {X 0,Y 453.762,Z 231.964,A -85,B 0,C 180,E1 -8457.335,E2 -8457.335} C_VEL
LIN {X 0,Y 453.82,Z 231.957,A -85,B 0,C 180,E1 -8459.999,E2 -8459.999} C_VEL
LIN {X 0,Y 453.76,Z 231.964,A -85,B 0,C 180,E1 -8462.662,E2 -8462.662} C_VEL
LIN {X 0,Y 453.672,Z 231.977,A -85,B 0,C 180,E1 -8466.224,E2 -8466.224} C_VEL
LIN {X 0,Y 453.585,Z 231.987,A -85,B 0,C 180,E1 -8468.912,E2 -8468.912} C_VEL
LIN {X 0,Y 453.476,Z 232.005,A -85,B 0,C 180,E1 -8471.622,E2 -8471.622} C_VEL
LIN {X 0,Y 453.229,Z 232.034,A -85,B 0,C 180,E1 -8473.448,E2 -8473.448} C_VEL
LIN {X 0,Y 453.167,Z 234.596,A -85,B 0,C 180,E1 -8476.208,E2 -8476.208} C_VEL
LIN {X 0,Y 453.093,Z 237.391,A -85,B 0,C 180,E1 -8479.008,E2 -8479.008} C_VEL
LIN {X 0,Y 452.968,Z 240.302,A -85,B 0,C 180,E1 -8481.86,E2 -8481.86} C_VEL
LIN {X 0,Y 452.917,Z 243.302,A -85,B 0,C 180,E1 -8484.767,E2 -8484.767} C_VEL
LIN {X 0,Y 452.846,Z 246.43,A -85,B 0,C 180,E1 -8487.797,E2 -8487.797} C_VEL
LIN {X 0,Y 452.784,Z 250.16,A -85,B 0,C 180,E1 -8491.238,E2 -8491.238} C_VEL
LIN {X 0,Y 456.154,Z 263.733,A -85,B 0,C 180,E1 -8491.802,E2 -8491.802} C_VEL
LIN {X 0,Y 456.657,Z 265.923,A -85,B 0,C 180,E1 -8491.908,E2 -8491.908} C_VEL
LIN {X 0,Y 456.318,Z 277.974,A -85,B 0,C 180,E1 -8492.499,E2 -8492.499} C_VEL
LIN {X 0,Y 455.819,Z 288.738,A -85,B 0,C 180,E1 -8493.183,E2 -8493.183} C_VEL
LIN {X 0,Y 455.329,Z 299.179,A -85,B 0,C 180,E1 -8494.02,E2 -8494.02} C_VEL
LIN {X 0,Y 454.817,Z 309.252,A -85,B 0,C 180,E1 -8495.019,E2 -8495.019} C_VEL
LIN {X 0,Y 454.249,Z 318.909,A -85,B 0,C 180,E1 -8496.211,E2 -8496.211} C_VEL
LIN {X 0,Y 453.761,Z 327.217,A -85,B 0,C 180,E1 -8497.477,E2 -8497.477} C_VEL
LIN {X 0,Y 453.421,Z 333.921,A -85,B 0,C 180,E1 -8498.736,E2 -8498.736} C_VEL
LIN {X 0,Y 453.071,Z 339.378,A -85,B 0,C 180,E1 -8500,E2 -8500} C_VEL
LIN {X 0,Y 452.917,Z 343.663,A -85,B 0,C 180,E1 -8501.247,E2 -8501.247} C_VEL
LIN {X 0,Y 452.764,Z 346.945,A -85,B 0,C 180,E1 -8502.469,E2 -8502.469} C_VEL
LIN {X 0,Y 452.695,Z 348.394,A -85,B 0,C 180,E1 -8503.143,E2 -8503.143} C_VEL
LIN {X 0,Y 452.552,Z 350.465,A -85,B 0,C 180,E1 -8504.41,E2 -8504.41} C_VEL
LIN {X 0,Y 452.487,Z 351.706,A -85,B 0,C 180,E1 -8505.659,E2 -8505.659} C_VEL
LIN {X 0,Y 452.458,Z 352.131,A -85,B 0,C 180,E1 -8506.887,E2 -8506.887} C_VEL
LIN {X 0,Y 452.453,Z 351.756,A -85,B 0,C 180,E1 -8508.207,E2 -8508.207} C_VEL
LIN {X 0,Y 452.518,Z 350.482,A -85,B 0,C 180,E1 -8509.55,E2 -8509.55} C_VEL
LIN {X 0,Y 452.641,Z 348.223,A -85,B 0,C 180,E1 -8510.923,E2 -8510.923} C_VEL
LIN {X 0,Y 452.79,Z 344.84,A -85,B 0,C 180,E1 -8512.332,E2 -8512.332} C_VEL
LIN {X 0,Y 453.051,Z 339.769,A -85,B 0,C 180,E1 -8513.881,E2 -8513.881} C_VEL
LIN {X 0,Y 453.325,Z 333.948,A -85,B 0,C 180,E1 -8515.249,E2 -8515.249} C_VEL
LIN {X 0,Y 453.672,Z 327.532,A -85,B 0,C 180,E1 -8516.463,E2 -8516.463} C_VEL
LIN {X 0,Y 454.131,Z 319.295,A -85,B 0,C 180,E1 -8517.731,E2 -8517.731} C_VEL
LIN {X 0,Y 454.625,Z 309.616,A -85,B 0,C 180,E1 -8518.94,E2 -8518.94} C_VEL
LIN {X 0,Y 455.099,Z 300.643,A -85,B 0,C 180,E1 -8519.855,E2 -8519.855} C_VEL
LIN {X 0,Y 455.616,Z 290.837,A -85,B 0,C 180,E1 -8520.677,E2 -8520.677} C_VEL
LIN {X 0,Y 456.082,Z 279,A -85,B 0,C 180,E1 -8521.466,E2 -8521.466} C_VEL
LIN {X 0,Y 456.514,Z 266.406,A -85,B 0,C 180,E1 -8522.098,E2 -8522.098} C_VEL
LIN {X 0,Y 454.104,Z 254.647,A -85,B 0,C 180,E1 -8522.617,E2 -8522.617} C_VEL
LIN {X 0,Y 452.731,Z 248.936,A -85,B 0,C 180,E1 -8522.84,E2 -8522.84} C_VEL
LIN {X 0,Y 452.723,Z 245.227,A -85,B 0,C 180,E1 -8526.196,E2 -8526.196} C_VEL
LIN {X 0,Y 452.764,Z 242.083,A -85,B 0,C 180,E1 -8529.084,E2 -8529.084} C_VEL
LIN {X 0,Y 452.742,Z 241.324,A -85,B 0,C 180,E1 -8529.779,E2 -8529.779} C_VEL
LIN {X 0,Y 452.089,Z 240.607,A -85,B 0,C 180,E1 -8530.516,E2 -8530.516} C_VEL
LIN {X 0,Y 449.248,Z 239.59,A -85,B 0,C 180,E1 -8531.717,E2 -8531.717} C_VEL
LIN {X 0,Y 446.859,Z 238.799,A -85,B 0,C 180,E1 -8532.686,E2 -8532.686} C_VEL
LIN {X 0,Y 445.862,Z 238.112,A -85,B 0,C 180,E1 -8533.433,E2 -8533.433} C_VEL
LIN {X 0,Y 445.797,Z 237.855,A -85,B 0,C 180,E1 -8533.686,E2 -8533.686} C_VEL
LIN {X 0,Y 445.864,Z 235.055,A -85,B 0,C 180,E1 -8536.324,E2 -8536.324} C_VEL
LIN {X 0,Y 445.958,Z 233.133,A -85,B 0,C 180,E1 -8538.179,E2 -8538.179} C_VEL
LIN {X 0,Y 446.298,Z 232.895,A -85,B 0,C 180,E1 -8540.94,E2 -8540.94} C_VEL
LIN {X 0,Y 446.623,Z 232.853,A -85,B 0,C 180,E1 -8543.677,E2 -8543.677} C_VEL
LIN {X 0,Y 446.694,Z 232.845,A -85,B 0,C 180,E1 -8547.295,E2 -8547.295} C_VEL
LIN {X 0,Y 446.778,Z 232.832,A -85,B 0,C 180,E1 -8550,E2 -8550} C_VEL
LIN {X 0,Y 446.695,Z 232.843,A -85,B 0,C 180,E1 -8552.706,E2 -8552.706} C_VEL
LIN {X 0,Y 446.633,Z 232.85,A -85,B 0,C 180,E1 -8556.324,E2 -8556.324} C_VEL
LIN {X 0,Y 446.524,Z 232.868,A -85,B 0,C 180,E1 -8559.056,E2 -8559.056} C_VEL
LIN {X 0,Y 446.518,Z 232.867,A -85,B 0,C 180,E1 -8562.73,E2 -8562.73} C_VEL
LIN {X 0,Y 446.475,Z 232.872,A -85,B 0,C 180,E1 -8566.46,E2 -8566.46} C_VEL
LIN {X 0,Y 446.456,Z 232.875,A -85,B 0,C 180,E1 -8569.304,E2 -8569.304} C_VEL
LIN {X 0,Y 446.427,Z 232.877,A -85,B 0,C 180,E1 -8572.2,E2 -8572.2} C_VEL
LIN {X 0,Y 446.459,Z 232.874,A -85,B 0,C 180,E1 -8575.153,E2 -8575.153} C_VEL
LIN {X 0,Y 446.471,Z 232.872,A -85,B 0,C 180,E1 -8578.18,E2 -8578.18} C_VEL
LIN {X 0,Y 446.407,Z 232.879,A -85,B 0,C 180,E1 -8581.777,E2 -8581.777} C_VEL
LIN {X 0,Y 446.419,Z 232.879,A -85,B 0,C 180,E1 -8584.524,E2 -8584.524} C_VEL
LIN {X 0,Y 446.427,Z 232.877,A -85,B 0,C 180,E1 -8588.085,E2 -8588.085} C_VEL
LIN {X 0,Y 446.437,Z 232.878,A -85,B 0,C 180,E1 -8590.922,E2 -8590.922} C_VEL
LIN {X 0,Y 446.436,Z 232.876,A -85,B 0,C 180,E1 -8593.842,E2 -8593.842} C_VEL
LIN {X 0,Y 446.438,Z 232.877,A -85,B 0,C 180,E1 -8596.399,E2 -8596.399} C_VEL
LIN {X 0,Y 446.461,Z 232.873,A -85,B 0,C 180,E1 -8599.807,E2 -8599.807} C_VEL
LIN {X 0,Y 446.427,Z 232.879,A -85,B 0,C 180,E1 -8602.126,E2 -8602.126} C_VEL
LIN {X 0,Y 446.424,Z 232.877,A -85,B 0,C 180,E1 -8605.479,E2 -8605.479} C_VEL
LIN {X 0,Y 446.415,Z 232.88,A -85,B 0,C 180,E1 -8608.702,E2 -8608.702} C_VEL
LIN {X 0,Y 446.48,Z 232.872,A -85,B 0,C 180,E1 -8611.823,E2 -8611.823} C_VEL
LIN {X 0,Y 446.454,Z 232.874,A -85,B 0,C 180,E1 -8614.85,E2 -8614.85} C_VEL
LIN {X 0,Y 446.446,Z 232.876,A -85,B 0,C 180,E1 -8618.247,E2 -8618.247} C_VEL
LIN {X 0,Y 446.456,Z 232.874,A -85,B 0,C 180,E1 -8621.651,E2 -8621.651} C_VEL
LIN {X 0,Y 446.507,Z 232.868,A -85,B 0,C 180,E1 -8624.482,E2 -8624.482} C_VEL
LIN {X 0,Y 446.517,Z 232.867,A -85,B 0,C 180,E1 -8628.195,E2 -8628.195} C_VEL
LIN {X 0,Y 446.533,Z 232.862,A -85,B 0,C 180,E1 -8630.946,E2 -8630.946} C_VEL
LIN {X 0,Y 446.642,Z 232.851,A -85,B 0,C 180,E1 -8633.678,E2 -8633.678} C_VEL
LIN {X 0,Y 446.692,Z 232.844,A -85,B 0,C 180,E1 -8637.296,E2 -8637.296} C_VEL
LIN {X 0,Y 446.795,Z 232.833,A -85,B 0,C 180,E1 -8640.002,E2 -8640.002} C_VEL
LIN {X 0,Y 446.692,Z 232.843,A -85,B 0,C 180,E1 -8642.707,E2 -8642.707} C_VEL
LIN {X 0,Y 446.623,Z 232.851,A -85,B 0,C 180,E1 -8646.325,E2 -8646.325} C_VEL
LIN {X 0,Y 446.524,Z 232.865,A -85,B 0,C 180,E1 -8649.971,E2 -8649.971} C_VEL
LIN {X 0,Y 446.526,Z 232.863,A -85,B 0,C 180,E1 -8652.731,E2 -8652.731} C_VEL
LIN {X 0,Y 446.502,Z 232.867,A -85,B 0,C 180,E1 -8656.229,E2 -8656.229} C_VEL
LIN {X 0,Y 446.475,Z 232.873,A -85,B 0,C 180,E1 -8659.304,E2 -8659.304} C_VEL
LIN {X 0,Y 446.423,Z 232.877,A -85,B 0,C 180,E1 -8662.201,E2 -8662.201} C_VEL
LIN {X 0,Y 446.443,Z 232.877,A -85,B 0,C 180,E1 -8665.154,E2 -8665.154} C_VEL
LIN {X 0,Y 446.491,Z 232.868,A -85,B 0,C 180,E1 -8668.179,E2 -8668.179} C_VEL
LIN {X 0,Y 446.424,Z 232.878,A -85,B 0,C 180,E1 -8671.775,E2 -8671.775} C_VEL
LIN {X 0,Y 446.429,Z 232.876,A -85,B 0,C 180,E1 -8674.524,E2 -8674.524} C_VEL
LIN {X 0,Y 446.421,Z 232.88,A -85,B 0,C 180,E1 -8678.08,E2 -8678.08} C_VEL
LIN {X 0,Y 446.433,Z 232.878,A -85,B 0,C 180,E1 -8680.918,E2 -8680.918} C_VEL
LIN {X 0,Y 446.405,Z 232.878,A -85,B 0,C 180,E1 -8683.847,E2 -8683.847} C_VEL
LIN {X 0,Y 446.403,Z 232.879,A -85,B 0,C 180,E1 -8686.404,E2 -8686.404} C_VEL
LIN {X 0,Y 446.475,Z 233.045,A -85,B 0,C 180,E1 -8688.161,E2 -8688.161} C_VEL
LIN {X 0,Y 447.583,Z 239.132,A -85,B 0,C 180,E1 -8691.091,E2 -8691.091} C_VEL
LIN {X 0,Y 448.389,Z 244.286,A -85,B 0,C 180,E1 -8693.444,E2 -8693.444} C_VEL
LIN {X 0,Y 448.327,Z 249.471,A -85,B 0,C 180,E1 -8695.643,E2 -8695.643} C_VEL
LIN {X 0,Y 447.811,Z 257.273,A -85,B 0,C 180,E1 -8698.808,E2 -8698.808} C_VEL
LIN {X 0,Y 447.266,Z 266.457,A -85,B 0,C 180,E1 -8702.384,E2 -8702.384} C_VEL
LIN {X 0,Y 446.892,Z 274.362,A -85,B 0,C 180,E1 -8705.371,E2 -8705.371} C_VEL
LIN {X 0,Y 446.535,Z 283.884,A -85,B 0,C 180,E1 -8708.777,E2 -8708.777} C_VEL
LIN {X 0,Y 446.179,Z 293.26,A -85,B 0,C 180,E1 -8712.112,E2 -8712.112} C_VEL
LIN {X 0,Y 446.013,Z 298.069,A -85,B 0,C 180,E1 -8713.818,E2 -8713.818} C_VEL
LIN {X 0,Y 448.465,Z 313.038,A -85,B 0,C 180,E1 -8714.343,E2 -8714.343} C_VEL
LIN {X 0,Y 449.421,Z 320.944,A -85,B 0,C 180,E1 -8714.699,E2 -8714.699} C_VEL
LIN {X 0,Y 448.96,Z 331.979,A -85,B 0,C 180,E1 -8715.263,E2 -8715.263} C_VEL
LIN {X 0,Y 448.369,Z 343.866,A -85,B 0,C 180,E1 -8716.054,E2 -8716.054} C_VEL
LIN {X 0,Y 447.802,Z 354.857,A -85,B 0,C 180,E1 -8716.993,E2 -8716.993} C_VEL
LIN {X 0,Y 447.293,Z 364.291,A -85,B 0,C 180,E1 -8717.983,E2 -8717.983} C_VEL
LIN {X 0,Y 446.682,Z 373.179,A -85,B 0,C 180,E1 -8719.116,E2 -8719.116} C_VEL
LIN {X 0,Y 446.262,Z 381.866,A -85,B 0,C 180,E1 -8720.481,E2 -8720.481} C_VEL
LIN {X 0,Y 445.887,Z 388.808,A -85,B 0,C 180,E1 -8721.844,E2 -8721.844} C_VEL
LIN {X 0,Y 445.653,Z 394.379,A -85,B 0,C 180,E1 -8723.207,E2 -8723.207} C_VEL
LIN {X 0,Y 445.542,Z 398.749,A -85,B 0,C 180,E1 -8724.569,E2 -8724.569} C_VEL
LIN {X 0,Y 445.429,Z 401.06,A -85,B 0,C 180,E1 -8725.475,E2 -8725.475} C_VEL
LIN {X 0,Y 445.398,Z 402.936,A -85,B 0,C 180,E1 -8726.381,E2 -8726.381} C_VEL
LIN {X 0,Y 445.424,Z 404.346,A -85,B 0,C 180,E1 -8727.286,E2 -8727.286} C_VEL
LIN {X 0,Y 445.357,Z 405.958,A -85,B 0,C 180,E1 -8729.095,E2 -8729.095} C_VEL
LIN {X 0,Y 445.351,Z 406.173,A -85,B 0,C 180,E1 -8730,E2 -8730} C_VEL
LIN {X 0,Y 445.357,Z 405.953,A -85,B 0,C 180,E1 -8730.904,E2 -8730.904} C_VEL
LIN {X 0,Y 445.424,Z 404.333,A -85,B 0,C 180,E1 -8732.713,E2 -8732.713} C_VEL
LIN {X 0,Y 445.398,Z 402.915,A -85,B 0,C 180,E1 -8733.618,E2 -8733.618} C_VEL
LIN {X 0,Y 445.501,Z 399.949,A -85,B 0,C 180,E1 -8734.977,E2 -8734.977} C_VEL
LIN {X 0,Y 445.59,Z 395.552,A -85,B 0,C 180,E1 -8736.451,E2 -8736.451} C_VEL
LIN {X 0,Y 445.804,Z 389.758,A -85,B 0,C 180,E1 -8737.928,E2 -8737.928} C_VEL
LIN {X 0,Y 446.183,Z 383.025,A -85,B 0,C 180,E1 -8739.291,E2 -8739.291} C_VEL
LIN {X 0,Y 446.609,Z 374.669,A -85,B 0,C 180,E1 -8740.655,E2 -8740.655} C_VEL
LIN {X 0,Y 447.175,Z 366.118,A -85,B 0,C 180,E1 -8741.789,E2 -8741.789} C_VEL
LIN {X 0,Y 447.711,Z 356.343,A -85,B 0,C 180,E1 -8742.849,E2 -8742.849} C_VEL
LIN {X 0,Y 448.217,Z 345.119,A -85,B 0,C 180,E1 -8743.834,E2 -8743.834} C_VEL
LIN {X 0,Y 448.845,Z 333.708,A -85,B 0,C 180,E1 -8744.624,E2 -8744.624} C_VEL
LIN {X 0,Y 449.376,Z 322.011,A -85,B 0,C 180,E1 -8745.244,E2 -8745.244} C_VEL
LIN {X 0,Y 449.006,Z 316.569,A -85,B 0,C 180,E1 -8745.494,E2 -8745.494} C_VEL
LIN {X 0,Y 446.694,Z 302.496,A -85,B 0,C 180,E1 -8746.032,E2 -8746.032} C_VEL
LIN {X 0,Y 446.008,Z 297.716,A -85,B 0,C 180,E1 -8746.181,E2 -8746.181} C_VEL
LIN {X 0,Y 446.329,Z 288.731,A -85,B 0,C 180,E1 -8749.309,E2 -8749.309} C_VEL
LIN {X 0,Y 446.588,Z 279.183,A -85,B 0,C 180,E1 -8752.678,E2 -8752.678} C_VEL
LIN {X 0,Y 446.902,Z 271.077,A -85,B 0,C 180,E1 -8755.623,E2 -8755.623} C_VEL
LIN {X 0,Y 447.35,Z 262.907,A -85,B 0,C 180,E1 -8758.711,E2 -8758.711} C_VEL
LIN {X 0,Y 447.86,Z 254.018,A -85,B 0,C 180,E1 -8762.244,E2 -8762.244} C_VEL
LIN {X 0,Y 448.416,Z 246.415,A -85,B 0,C 180,E1 -8765.443,E2 -8765.443} C_VEL
LIN {X 0,Y 448.297,Z 243.15,A -85,B 0,C 180,E1 -8766.913,E2 -8766.913} C_VEL
LIN {X 0,Y 447.112,Z 236.617,A -85,B 0,C 180,E1 -8770.125,E2 -8770.125} C_VEL
LIN {X 0,Y 446.417,Z 232.883,A -85,B 0,C 180,E1 -8772.2,E2 -8772.2} C_VEL
LIN {X 0,Y 446.455,Z 232.875,A -85,B 0,C 180,E1 -8775.102,E2 -8775.102} C_VEL
LIN {X 0,Y 446.437,Z 232.877,A -85,B 0,C 180,E1 -8778.609,E2 -8778.609} C_VEL
LIN {X 0,Y 446.476,Z 232.874,A -85,B 0,C 180,E1 -8780.975,E2 -8780.975} C_VEL
LIN {X 0,Y 446.419,Z 232.88,A -85,B 0,C 180,E1 -8784.373,E2 -8784.373} C_VEL
LIN {X 0,Y 446.422,Z 232.879,A -85,B 0,C 180,E1 -8787.637,E2 -8787.637} C_VEL
LIN {X 0,Y 446.449,Z 232.874,A -85,B 0,C 180,E1 -8790.789,E2 -8790.789} C_VEL
LIN {X 0,Y 446.477,Z 232.871,A -85,B 0,C 180,E1 -8793.847,E2 -8793.847} C_VEL
LIN {X 0,Y 446.429,Z 232.877,A -85,B 0,C 180,E1 -8796.822,E2 -8796.822} C_VEL
LIN {X 0,Y 446.444,Z 232.873,A -85,B 0,C 180,E1 -8799.736,E2 -8799.736} C_VEL
LIN {X 0,Y 446.462,Z 232.872,A -85,B 0,C 180,E1 -8802.596,E2 -8802.596} C_VEL
LIN {X 0,Y 446.468,Z 232.873,A -85,B 0,C 180,E1 -8805.411,E2 -8805.411} C_VEL
LIN {X 0,Y 446.515,Z 232.867,A -85,B 0,C 180,E1 -8808.192,E2 -8808.192} C_VEL
LIN {X 0,Y 446.597,Z 232.856,A -85,B 0,C 180,E1 -8811.856,E2 -8811.856} C_VEL
LIN {X 0,Y 446.643,Z 232.851,A -85,B 0,C 180,E1 -8814.581,E2 -8814.581} C_VEL
LIN {X 0,Y 446.706,Z 232.843,A -85,B 0,C 180,E1 -8817.293,E2 -8817.293} C_VEL
LIN {X 0,Y 446.79,Z 232.832,A -85,B 0,C 180,E1 -8819.998,E2 -8819.998} C_VEL
LIN {X 0,Y 446.704,Z 232.843,A -85,B 0,C 180,E1 -8822.704,E2 -8822.704} C_VEL
LIN {X 0,Y 446.641,Z 232.853,A -85,B 0,C 180,E1 -8826.322,E2 -8826.322} C_VEL
LIN {X 0,Y 446.53,Z 232.866,A -85,B 0,C 180,E1 -8829.054,E2 -8829.054} C_VEL
LIN {X 0,Y 446.416,Z 232.885,A -85,B 0,C 180,E1 -8831.808,E2 -8831.808} C_VEL
LIN {X 0,Y 446.153,Z 232.976,A -85,B 0,C 180,E1 -8833.666,E2 -8833.666} C_VEL
LIN {X 0,Y 446.1,Z 235.727,A -85,B 0,C 180,E1 -8836.472,E2 -8836.472} C_VEL
LIN {X 0,Y 446.013,Z 238.54,A -85,B 0,C 180,E1 -8839.322,E2 -8839.322} C_VEL
LIN {X 0,Y 445.896,Z 241.517,A -85,B 0,C 180,E1 -8842.225,E2 -8842.225} C_VEL
LIN {X 0,Y 445.838,Z 244.527,A -85,B 0,C 180,E1 -8845.188,E2 -8845.188} C_VEL
LIN {X 0,Y 445.758,Z 247.653,A -85,B 0,C 180,E1 -8848.227,E2 -8848.227} C_VEL
LIN {X 0,Y 445.714,Z 250.507,A -85,B 0,C 180,E1 -8850.957,E2 -8850.957} C_VEL
LIN {X 0,Y 449.255,Z 264.583,A -85,B 0,C 180,E1 -8851.574,E2 -8851.574} C_VEL
LIN {X 0,Y 449.819,Z 269.013,A -85,B 0,C 180,E1 -8851.79,E2 -8851.79} C_VEL
LIN {X 0,Y 449.323,Z 281.398,A -85,B 0,C 180,E1 -8852.441,E2 -8852.441} C_VEL
LIN {X 0,Y 448.809,Z 292.746,A -85,B 0,C 180,E1 -8853.233,E2 -8853.233} C_VEL
LIN {X 0,Y 448.213,Z 303.85,A -85,B 0,C 180,E1 -8854.214,E2 -8854.214} C_VEL
LIN {X 0,Y 447.631,Z 313.522,A -85,B 0,C 180,E1 -8855.273,E2 -8855.273} C_VEL
LIN {X 0,Y 447.169,Z 321.835,A -85,B 0,C 180,E1 -8856.389,E2 -8856.389} C_VEL
LIN {X 0,Y 446.701,Z 329.046,A -85,B 0,C 180,E1 -8857.562,E2 -8857.562} C_VEL
LIN {X 0,Y 446.259,Z 336.367,A -85,B 0,C 180,E1 -8859.044,E2 -8859.044} C_VEL
LIN {X 0,Y 445.952,Z 342.167,A -85,B 0,C 180,E1 -8860.542,E2 -8860.542} C_VEL
LIN {X 0,Y 445.707,Z 346.883,A -85,B 0,C 180,E1 -8862.175,E2 -8862.175} C_VEL
LIN {X 0,Y 445.504,Z 350.337,A -85,B 0,C 180,E1 -8863.954,E2 -8863.954} C_VEL
LIN {X 0,Y 445.402,Z 351.821,A -85,B 0,C 180,E1 -8865.236,E2 -8865.236} C_VEL
LIN {X 0,Y 445.371,Z 352.514,A -85,B 0,C 180,E1 -8866.539,E2 -8866.539} C_VEL
LIN {X 0,Y 445.361,Z 352.38,A -85,B 0,C 180,E1 -8867.872,E2 -8867.872} C_VEL
LIN {X 0,Y 445.442,Z 350.77,A -85,B 0,C 180,E1 -8869.694,E2 -8869.694} C_VEL
LIN {X 0,Y 445.571,Z 348.835,A -85,B 0,C 180,E1 -8870.883,E2 -8870.883} C_VEL
LIN {X 0,Y 445.772,Z 344.653,A -85,B 0,C 180,E1 -8872.629,E2 -8872.629} C_VEL
LIN {X 0,Y 445.992,Z 340.407,A -85,B 0,C 180,E1 -8873.921,E2 -8873.921} C_VEL
LIN {X 0,Y 446.264,Z 335.016,A -85,B 0,C 180,E1 -8875.227,E2 -8875.227} C_VEL
LIN {X 0,Y 446.661,Z 328.055,A -85,B 0,C 180,E1 -8876.585,E2 -8876.585} C_VEL
LIN {X 0,Y 447.168,Z 319.519,A -85,B 0,C 180,E1 -8877.916,E2 -8877.916} C_VEL
LIN {X 0,Y 447.692,Z 309.841,A -85,B 0,C 180,E1 -8879.14,E2 -8879.14} C_VEL
LIN {X 0,Y 448.271,Z 299.977,A -85,B 0,C 180,E1 -8880.148,E2 -8880.148} C_VEL
LIN {X 0,Y 448.809,Z 288.931,A -85,B 0,C 180,E1 -8881.052,E2 -8881.052} C_VEL
LIN {X 0,Y 449.326,Z 276.703,A -85,B 0,C 180,E1 -8881.837,E2 -8881.837} C_VEL
LIN {X 0,Y 449.579,Z 266.303,A -85,B 0,C 180,E1 -8882.35,E2 -8882.35} C_VEL
LIN {X 0,Y 446.678,Z 253.608,A -85,B 0,C 180,E1 -8882.916,E2 -8882.916} C_VEL
LIN {X 0,Y 445.666,Z 249.334,A -85,B 0,C 180,E1 -8883.072,E2 -8883.072} C_VEL
LIN {X 0,Y 445.655,Z 245.958,A -85,B 0,C 180,E1 -8886.152,E2 -8886.152} C_VEL
LIN {X 0,Y 445.691,Z 243.156,A -85,B 0,C 180,E1 -8888.736,E2 -8888.736} C_VEL
LIN {X 0,Y 445.799,Z 240.038,A -85,B 0,C 180,E1 -8891.622,E2 -8891.622} C_VEL
LIN {X 0,Y 445.797,Z 237.855,A -85,B 0,C 180,E1 -8893.686,E2 -8893.686} C_VEL
LIN {X 0,Y 445.184,Z 237.142,A -85,B 0,C 180,E1 -8894.434,E2 -8894.434} C_VEL
LIN {X 0,Y 442.392,Z 236.147,A -85,B 0,C 180,E1 -8895.655,E2 -8895.655} C_VEL
LIN {X 0,Y 440.004,Z 235.376,A -85,B 0,C 180,E1 -8896.64,E2 -8896.64} C_VEL
LIN {X 0,Y 438.977,Z 234.705,A -85,B 0,C 180,E1 -8897.399,E2 -8897.399} C_VEL
LIN {X 0,Y 438.894,Z 234.45,A -85,B 0,C 180,E1 -8897.655,E2 -8897.655} C_VEL
LIN {X 0,Y 438.972,Z 233.809,A -85,B 0,C 180,E1 -8898.924,E2 -8898.924} C_VEL
LIN {X 0,Y 439.509,Z 233.738,A -85,B 0,C 180,E1 -8902.469,E2 -8902.469} C_VEL
LIN {X 0,Y 439.607,Z 233.725,A -85,B 0,C 180,E1 -8904.496,E2 -8904.496} C_VEL
LIN {X 0,Y 439.62,Z 233.724,A -85,B 0,C 180,E1 -8908.168,E2 -8908.168} C_VEL
LIN {X 0,Y 439.748,Z 233.708,A -85,B 0,C 180,E1 -8910.001,E2 -8910.001} C_VEL
LIN {X 0,Y 439.642,Z 233.722,A -85,B 0,C 180,E1 -8912.749,E2 -8912.749} C_VEL
LIN {X 0,Y 439.604,Z 233.726,A -85,B 0,C 180,E1 -8916.426,E2 -8916.426} C_VEL
LIN {X 0,Y 439.486,Z 233.743,A -85,B 0,C 180,E1 -8919.202,E2 -8919.202} C_VEL
LIN {X 0,Y 439.488,Z 233.743,A -85,B 0,C 180,E1 -8922.727,E2 -8922.727} C_VEL
LIN {X 0,Y 439.432,Z 233.748,A -85,B 0,C 180,E1 -8926.35,E2 -8926.35} C_VEL
LIN {X 0,Y 439.421,Z 233.749,A -85,B 0,C 180,E1 -8929.626,E2 -8929.626} C_VEL
LIN {X 0,Y 439.367,Z 233.757,A -85,B 0,C 180,E1 -8932.576,E2 -8932.576} C_VEL
LIN {X 0,Y 439.4,Z 233.752,A -85,B 0,C 180,E1 -8935.586,E2 -8935.586} C_VEL
LIN {X 0,Y 439.404,Z 233.753,A -85,B 0,C 180,E1 -8938.675,E2 -8938.675} C_VEL
LIN {X 0,Y 439.358,Z 233.757,A -85,B 0,C 180,E1 -8942.032,E2 -8942.032} C_VEL
LIN {X 0,Y 439.384,Z 233.753,A -85,B 0,C 180,E1 -8945.342,E2 -8945.342} C_VEL
LIN {X 0,Y 439.388,Z 233.756,A -85,B 0,C 180,E1 -8948.595,E2 -8948.595} C_VEL
LIN {X 0,Y 439.395,Z 233.752,A -85,B 0,C 180,E1 -8951.261,E2 -8951.261} C_VEL
LIN {X 0,Y 439.401,Z 233.754,A -85,B 0,C 180,E1 -8954.73,E2 -8954.73} C_VEL
LIN {X 0,Y 439.404,Z 233.751,A -85,B 0,C 180,E1 -8957.799,E2 -8957.799} C_VEL
LIN {X 0,Y 439.444,Z 233.748,A -85,B 0,C 180,E1 -8960.232,E2 -8960.232} C_VEL
LIN {X 0,Y 439.37,Z 233.755,A -85,B 0,C 180,E1 -8963.715,E2 -8963.715} C_VEL
LIN {X 0,Y 439.369,Z 233.754,A -85,B 0,C 180,E1 -8967.056,E2 -8967.056} C_VEL
LIN {X 0,Y 439.392,Z 233.756,A -85,B 0,C 180,E1 -8970.277,E2 -8970.277} C_VEL
LIN {X 0,Y 439.429,Z 233.747,A -85,B 0,C 180,E1 -8973.591,E2 -8973.591} C_VEL
LIN {X 0,Y 439.384,Z 233.755,A -85,B 0,C 180,E1 -8976.431,E2 -8976.431} C_VEL
LIN {X 0,Y 439.386,Z 233.752,A -85,B 0,C 180,E1 -8979.399,E2 -8979.399} C_VEL
LIN {X 0,Y 439.43,Z 233.749,A -85,B 0,C 180,E1 -8982.311,E2 -8982.311} C_VEL
LIN {X 0,Y 439.447,Z 233.745,A -85,B 0,C 180,E1 -8985.176,E2 -8985.176} C_VEL
LIN {X 0,Y 439.483,Z 233.744,A -85,B 0,C 180,E1 -8988.003,E2 -8988.003} C_VEL
LIN {X 0,Y 439.504,Z 233.741,A -85,B 0,C 180,E1 -8991.727,E2 -8991.727} C_VEL
LIN {X 0,Y 439.621,Z 233.724,A -85,B 0,C 180,E1 -8994.497,E2 -8994.497} C_VEL
LIN {X 0,Y 439.636,Z 233.723,A -85,B 0,C 180,E1 -8998.169,E2 -8998.169} C_VEL
LIN {X 0,Y 439.765,Z 233.708,A -85,B 0,C 180,E1 -9000.002,E2 -9000.002} C_VEL
LIN {X 0,Y 439.642,Z 233.721,A -85,B 0,C 180,E1 -9002.75,E2 -9002.75} C_VEL
LIN {X 0,Y 439.595,Z 233.726,A -85,B 0,C 180,E1 -9006.427,E2 -9006.427} C_VEL
LIN {X 0,Y 439.499,Z 233.74,A -85,B 0,C 180,E1 -9009.203,E2 -9009.203} C_VEL
LIN {X 0,Y 439.47,Z 233.742,A -85,B 0,C 180,E1 -9012.939,E2 -9012.939} C_VEL
LIN {X 0,Y 439.453,Z 233.745,A -85,B 0,C 180,E1 -9016.35,E2 -9016.35} C_VEL
LIN {X 0,Y 439.408,Z 233.752,A -85,B 0,C 180,E1 -9019.627,E2 -9019.627} C_VEL
LIN {X 0,Y 439.369,Z 233.755,A -85,B 0,C 180,E1 -9022.577,E2 -9022.577} C_VEL
LIN {X 0,Y 439.392,Z 233.754,A -85,B 0,C 180,E1 -9025.587,E2 -9025.587} C_VEL
LIN {X 0,Y 439.423,Z 233.749,A -85,B 0,C 180,E1 -9028.674,E2 -9028.674} C_VEL
LIN {X 0,Y 439.374,Z 233.755,A -85,B 0,C 180,E1 -9032.031,E2 -9032.031} C_VEL
LIN {X 0,Y 439.398,Z 233.754,A -85,B 0,C 180,E1 -9035.34,E2 -9035.34} C_VEL
LIN {X 0,Y 439.384,Z 233.755,A -85,B 0,C 180,E1 -9038.596,E2 -9038.596} C_VEL
LIN {X 0,Y 439.395,Z 233.754,A -85,B 0,C 180,E1 -9041.257,E2 -9041.257} C_VEL
LIN {X 0,Y 439.405,Z 233.75,A -85,B 0,C 180,E1 -9044.73,E2 -9044.73} C_VEL
LIN {X 0,Y 439.43,Z 233.855,A -85,B 0,C 180,E1 -9047.799,E2 -9047.799} C_VEL
LIN {X 0,Y 440.593,Z 240.204,A -85,B 0,C 180,E1 -9050.913,E2 -9050.913} C_VEL
LIN {X 0,Y 441.401,Z 245.454,A -85,B 0,C 180,E1 -9053.355,E2 -9053.355} C_VEL
LIN {X 0,Y 441.37,Z 249.295,A -85,B 0,C 180,E1 -9055.024,E2 -9055.024} C_VEL
LIN {X 0,Y 440.971,Z 255.561,A -85,B 0,C 180,E1 -9057.64,E2 -9057.64} C_VEL
LIN {X 0,Y 440.428,Z 263.605,A -85,B 0,C 180,E1 -9060.877,E2 -9060.877} C_VEL
LIN {X 0,Y 440.023,Z 271.464,A -85,B 0,C 180,E1 -9063.945,E2 -9063.945} C_VEL
LIN {X 0,Y 439.632,Z 279.472,A -85,B 0,C 180,E1 -9066.942,E2 -9066.942} C_VEL
LIN {X 0,Y 439.31,Z 287.524,A -85,B 0,C 180,E1 -9069.882,E2 -9069.882} C_VEL
LIN {X 0,Y 439.004,Z 295.511,A -85,B 0,C 180,E1 -9072.772,E2 -9072.772} C_VEL
LIN {X 0,Y 438.946,Z 297.706,A -85,B 0,C 180,E1 -9073.563,E2 -9073.563} C_VEL
LIN {X 0,Y 441.247,Z 311.887,A -85,B 0,C 180,E1 -9074.052,E2 -9074.052} C_VEL
LIN {X 0,Y 442.507,Z 321.816,A -85,B 0,C 180,E1 -9074.513,E2 -9074.513} C_VEL
LIN {X 0,Y 441.968,Z 333.487,A -85,B 0,C 180,E1 -9075.142,E2 -9075.142} C_VEL
LIN {X 0,Y 441.361,Z 344.879,A -85,B 0,C 180,E1 -9075.946,E2 -9075.946} C_VEL
LIN {X 0,Y 440.737,Z 356.266,A -85,B 0,C 180,E1 -9076.963,E2 -9076.963} C_VEL
LIN {X 0,Y 440.199,Z 365.824,A -85,B 0,C 180,E1 -9078.021,E2 -9078.021} C_VEL
LIN {X 0,Y 439.594,Z 374.356,A -85,B 0,C 180,E1 -9079.172,E2 -9079.172} C_VEL
LIN {X 0,Y 439.155,Z 382.69,A -85,B 0,C 180,E1 -9080.558,E2 -9080.558} C_VEL
LIN {X 0,Y 438.755,Z 389.406,A -85,B 0,C 180,E1 -9081.943,E2 -9081.943} C_VEL
LIN {X 0,Y 438.53,Z 395.565,A -85,B 0,C 180,E1 -9083.558,E2 -9083.558} C_VEL
LIN {X 0,Y 438.436,Z 399.567,A -85,B 0,C 180,E1 -9084.942,E2 -9084.942} C_VEL
LIN {X 0,Y 438.303,Z 402.517,A -85,B 0,C 180,E1 -9086.322,E2 -9086.322} C_VEL
LIN {X 0,Y 438.352,Z 403.929,A -85,B 0,C 180,E1 -9087.243,E2 -9087.243} C_VEL
LIN {X 0,Y 438.27,Z 405.538,A -85,B 0,C 180,E1 -9089.081,E2 -9089.081} C_VEL
LIN {X 0,Y 438.291,Z 405.753,A -85,B 0,C 180,E1 -9089.999,E2 -9089.999} C_VEL
LIN {X 0,Y 438.27,Z 405.53,A -85,B 0,C 180,E1 -9090.918,E2 -9090.918} C_VEL
LIN {X 0,Y 438.352,Z 403.905,A -85,B 0,C 180,E1 -9092.756,E2 -9092.756} C_VEL
LIN {X 0,Y 438.304,Z 402.483,A -85,B 0,C 180,E1 -9093.677,E2 -9093.677} C_VEL
LIN {X 0,Y 438.436,Z 399.514,A -85,B 0,C 180,E1 -9095.057,E2 -9095.057} C_VEL
LIN {X 0,Y 438.509,Z 395.489,A -85,B 0,C 180,E1 -9096.441,E2 -9096.441} C_VEL
LIN {X 0,Y 438.754,Z 389.31,A -85,B 0,C 180,E1 -9098.056,E2 -9098.056} C_VEL
LIN {X 0,Y 439.143,Z 382.569,A -85,B 0,C 180,E1 -9099.441,E2 -9099.441} C_VEL
LIN {X 0,Y 439.594,Z 374.206,A -85,B 0,C 180,E1 -9100.827,E2 -9100.827} C_VEL
LIN {X 0,Y 440.194,Z 365.649,A -85,B 0,C 180,E1 -9101.978,E2 -9101.978} C_VEL
LIN {X 0,Y 440.738,Z 356.101,A -85,B 0,C 180,E1 -9103.032,E2 -9103.032} C_VEL
LIN {X 0,Y 441.302,Z 344.641,A -85,B 0,C 180,E1 -9104.055,E2 -9104.055} C_VEL
LIN {X 0,Y 441.954,Z 333.228,A -85,B 0,C 180,E1 -9104.857,E2 -9104.857} C_VEL
LIN {X 0,Y 442.503,Z 321.531,A -85,B 0,C 180,E1 -9105.487,E2 -9105.487} C_VEL
LIN {X 0,Y 440.863,Z 309.674,A -85,B 0,C 180,E1 -9106.025,E2 -9106.025} C_VEL
LIN {X 0,Y 438.91,Z 297.235,A -85,B 0,C 180,E1 -9106.453,E2 -9106.453} C_VEL
LIN {X 0,Y 439.259,Z 288.256,A -85,B 0,C 180,E1 -9109.632,E2 -9109.632} C_VEL
LIN {X 0,Y 439.56,Z 278.82,A -85,B 0,C 180,E1 -9113.061,E2 -9113.061} C_VEL
LIN {X 0,Y 439.923,Z 270.825,A -85,B 0,C 180,E1 -9116.054,E2 -9116.054} C_VEL
LIN {X 0,Y 440.357,Z 262.863,A -85,B 0,C 180,E1 -9119.128,E2 -9119.128} C_VEL
LIN {X 0,Y 440.862,Z 254.972,A -85,B 0,C 180,E1 -9122.337,E2 -9122.337} C_VEL
LIN {X 0,Y 441.342,Z 248.788,A -85,B 0,C 180,E1 -9124.978,E2 -9124.978} C_VEL
LIN {X 0,Y 441.409,Z 245.097,A -85,B 0,C 180,E1 -9126.638,E2 -9126.638} C_VEL
LIN {X 0,Y 440.236,Z 238.398,A -85,B 0,C 180,E1 -9129.978,E2 -9129.978} C_VEL
LIN {X 0,Y 439.384,Z 233.758,A -85,B 0,C 180,E1 -9132.626,E2 -9132.626} C_VEL
LIN {X 0,Y 439.403,Z 233.753,A -85,B 0,C 180,E1 -9135.27,E2 -9135.27} C_VEL
LIN {X 0,Y 439.4,Z 233.753,A -85,B 0,C 180,E1 -9138.741,E2 -9138.741} C_VEL
LIN {X 0,Y 439.393,Z 233.755,A -85,B 0,C 180,E1 -9141.604,E2 -9141.604} C_VEL
LIN {X 0,Y 439.399,Z 233.754,A -85,B 0,C 180,E1 -9144.843,E2 -9144.843} C_VEL
LIN {X 0,Y 439.373,Z 233.758,A -85,B 0,C 180,E1 -9148.138,E2 -9148.138} C_VEL
LIN {X 0,Y 439.432,Z 233.749,A -85,B 0,C 180,E1 -9151.597,E2 -9151.597} C_VEL
LIN {X 0,Y 439.405,Z 233.753,A -85,B 0,C 180,E1 -9154.414,E2 -9154.414} C_VEL
LIN {X 0,Y 439.364,Z 233.756,A -85,B 0,C 180,E1 -9157.423,E2 -9157.423} C_VEL
LIN {X 0,Y 439.44,Z 233.749,A -85,B 0,C 180,E1 -9160.661,E2 -9160.661} C_VEL
LIN {X 0,Y 439.461,Z 233.744,A -85,B 0,C 180,E1 -9164.223,E2 -9164.223} C_VEL
LIN {X 0,Y 439.481,Z 233.744,A -85,B 0,C 180,E1 -9168,E2 -9168} C_VEL
LIN {X 0,Y 439.545,Z 233.733,A -85,B 0,C 180,E1 -9171.725,E2 -9171.725} C_VEL
LIN {X 0,Y 439.619,Z 233.726,A -85,B 0,C 180,E1 -9174.494,E2 -9174.494} C_VEL
LIN {X 0,Y 439.632,Z 233.724,A -85,B 0,C 180,E1 -9178.166,E2 -9178.166} C_VEL
LIN {X 0,Y 439.761,Z 233.708,A -85,B 0,C 180,E1 -9179.998,E2 -9179.998} C_VEL
LIN {X 0,Y 439.651,Z 233.722,A -85,B 0,C 180,E1 -9182.747,E2 -9182.747} C_VEL
LIN {X 0,Y 439.613,Z 233.729,A -85,B 0,C 180,E1 -9186.424,E2 -9186.424} C_VEL
LIN {X 0,Y 439.49,Z 233.743,A -85,B 0,C 180,E1 -9189.2,E2 -9189.2} C_VEL
LIN {X 0,Y 439.289,Z 233.773,A -85,B 0,C 180,E1 -9192.605,E2 -9192.605} C_VEL
LIN {X 0,Y 439.104,Z 234.127,A -85,B 0,C 180,E1 -9193.889,E2 -9193.889} C_VEL
LIN {X 0,Y 439.025,Z 236.862,A -85,B 0,C 180,E1 -9196.745,E2 -9196.745} C_VEL
LIN {X 0,Y 438.937,Z 239.763,A -85,B 0,C 180,E1 -9199.646,E2 -9199.646} C_VEL
LIN {X 0,Y 438.832,Z 242.724,A -85,B 0,C 180,E1 -9202.602,E2 -9202.602} C_VEL
LIN {X 0,Y 438.765,Z 245.775,A -85,B 0,C 180,E1 -9205.623,E2 -9205.623} C_VEL
LIN {X 0,Y 438.687,Z 248.937,A -85,B 0,C 180,E1 -9208.723,E2 -9208.723} C_VEL
LIN {X 0,Y 438.649,Z 250.977,A -85,B 0,C 180,E1 -9210.687,E2 -9210.687} C_VEL
LIN {X 0,Y 442.286,Z 265.172,A -85,B 0,C 180,E1 -9211.324,E2 -9211.324} C_VEL
LIN {X 0,Y 442.991,Z 269.962,A -85,B 0,C 180,E1 -9211.568,E2 -9211.568} C_VEL
LIN {X 0,Y 442.478,Z 281.934,A -85,B 0,C 180,E1 -9212.212,E2 -9212.212} C_VEL
LIN {X 0,Y 441.945,Z 293.057,A -85,B 0,C 180,E1 -9212.999,E2 -9212.999} C_VEL
LIN {X 0,Y 441.32,Z 304.193,A -85,B 0,C 180,E1 -9213.996,E2 -9213.996} C_VEL
LIN {X 0,Y 440.683,Z 314.585,A -85,B 0,C 180,E1 -9215.158,E2 -9215.158} C_VEL
LIN {X 0,Y 440.153,Z 323.435,A -85,B 0,C 180,E1 -9216.396,E2 -9216.396} C_VEL
LIN {X 0,Y 439.628,Z 330.769,A -85,B 0,C 180,E1 -9217.648,E2 -9217.648} C_VEL
LIN {X 0,Y 439.188,Z 338.014,A -85,B 0,C 180,E1 -9219.19,E2 -9219.19} C_VEL
LIN {X 0,Y 438.912,Z 342.587,A -85,B 0,C 180,E1 -9220.426,E2 -9220.426} C_VEL
LIN {X 0,Y 438.701,Z 346.324,A -85,B 0,C 180,E1 -9221.693,E2 -9221.693} C_VEL
LIN {X 0,Y 438.599,Z 348.289,A -85,B 0,C 180,E1 -9222.517,E2 -9222.517} C_VEL
LIN {X 0,Y 438.433,Z 350.679,A -85,B 0,C 180,E1 -9223.836,E2 -9223.836} C_VEL
LIN {X 0,Y 438.322,Z 352.2,A -85,B 0,C 180,E1 -9225.132,E2 -9225.132} C_VEL
LIN {X 0,Y 438.294,Z 352.931,A -85,B 0,C 180,E1 -9226.41,E2 -9226.41} C_VEL
LIN {X 0,Y 438.274,Z 352.891,A -85,B 0,C 180,E1 -9227.663,E2 -9227.663} C_VEL
LIN {X 0,Y 438.319,Z 352.112,A -85,B 0,C 180,E1 -9228.9,E2 -9228.9} C_VEL
LIN {X 0,Y 438.428,Z 350.368,A -85,B 0,C 180,E1 -9230.3,E2 -9230.3} C_VEL
LIN {X 0,Y 438.578,Z 347.573,A -85,B 0,C 180,E1 -9231.736,E2 -9231.736} C_VEL
LIN {X 0,Y 438.771,Z 343.566,A -85,B 0,C 180,E1 -9233.21,E2 -9233.21} C_VEL
LIN {X 0,Y 439.128,Z 337.74,A -85,B 0,C 180,E1 -9234.82,E2 -9234.82} C_VEL
LIN {X 0,Y 439.513,Z 331.043,A -85,B 0,C 180,E1 -9236.249,E2 -9236.249} C_VEL
LIN {X 0,Y 440.041,Z 322.534,A -85,B 0,C 180,E1 -9237.697,E2 -9237.697} C_VEL
LIN {X 0,Y 440.622,Z 313.694,A -85,B 0,C 180,E1 -9238.911,E2 -9238.911} C_VEL
LIN {X 0,Y 441.111,Z 303.839,A -85,B 0,C 180,E1 -9240.009,E2 -9240.009} C_VEL
LIN {X 0,Y 441.785,Z 292.321,A -85,B 0,C 180,E1 -9241.034,E2 -9241.034} C_VEL
LIN {X 0,Y 442.261,Z 281.701,A -85,B 0,C 180,E1 -9241.787,E2 -9241.787} C_VEL
LIN {X 0,Y 442.78,Z 269.136,A -85,B 0,C 180,E1 -9242.466,E2 -9242.466} C_VEL
LIN {X 0,Y 441.935,Z 263.88,A -85,B 0,C 180,E1 -9242.73,E2 -9242.73} C_VEL
LIN {X 0,Y 438.748,Z 250.717,A -85,B 0,C 180,E1 -9243.288,E2 -9243.288} C_VEL
LIN {X 0,Y 438.612,Z 249.697,A -85,B 0,C 180,E1 -9243.343,E2 -9243.343} C_VEL
LIN {X 0,Y 438.6,Z 246.39,A -85,B 0,C 180,E1 -9246.385,E2 -9246.385} C_VEL
LIN {X 0,Y 438.612,Z 243.171,A -85,B 0,C 180,E1 -9249.36,E2 -9249.36} C_VEL
LIN {X 0,Y 438.715,Z 240.079,A -85,B 0,C 180,E1 -9252.28,E2 -9252.28} C_VEL
LIN {X 0,Y 438.757,Z 237.056,A -85,B 0,C 180,E1 -9255.151,E2 -9255.151} C_VEL
LIN {X 0,Y 438.894,Z 234.45,A -85,B 0,C 180,E1 -9257.655,E2 -9257.655} C_VEL
LIN {X 0,Y 438.256,Z 234.02,A -85,B 0,C 180,E1 -9258.418,E2 -9258.418} C_VEL
LIN {X 0,Y 435.551,Z 234.234,A -85,B 0,C 180,E1 -9259.667,E2 -9259.667} C_VEL
LIN {X 0,Y 433.3,Z 234.523,A -85,B 0,C 180,E1 -9260.678,E2 -9260.678} C_VEL
LIN {X 0,Y 432.384,Z 234.63,A -85,B 0,C 180,E1 -9261.456,E2 -9261.456} C_VEL
LIN {X 0,Y 432.336,Z 234.633,A -85,B 0,C 180,E1 -9261.719,E2 -9261.719} C_VEL
LIN {X 0,Y 432.582,Z 234.6,A -85,B 0,C 180,E1 -9264.406,E2 -9264.406} C_VEL
LIN {X 0,Y 432.59,Z 234.6,A -85,B 0,C 180,E1 -9268.139,E2 -9268.139} C_VEL
LIN {X 0,Y 432.718,Z 234.584,A -85,B 0,C 180,E1 -9270.001,E2 -9270.001} C_VEL
LIN {X 0,Y 432.591,Z 234.6,A -85,B 0,C 180,E1 -9272.794,E2 -9272.794} C_VEL
LIN {X 0,Y 432.559,Z 234.604,A -85,B 0,C 180,E1 -9276.531,E2 -9276.531} C_VEL
LIN {X 0,Y 432.43,Z 234.621,A -85,B 0,C 180,E1 -9279.354,E2 -9279.354} C_VEL
LIN {X 0,Y 432.429,Z 234.623,A -85,B 0,C 180,E1 -9282.813,E2 -9282.813} C_VEL
LIN {X 0,Y 432.397,Z 234.625,A -85,B 0,C 180,E1 -9286.48,E2 -9286.48} C_VEL
LIN {X 0,Y 432.368,Z 234.627,A -85,B 0,C 180,E1 -9289.959,E2 -9289.959} C_VEL
LIN {X 0,Y 432.316,Z 234.636,A -85,B 0,C 180,E1 -9292.965,E2 -9292.965} C_VEL
LIN {X 0,Y 432.355,Z 234.629,A -85,B 0,C 180,E1 -9296.033,E2 -9296.033} C_VEL
LIN {X 0,Y 432.33,Z 234.633,A -85,B 0,C 180,E1 -9299.189,E2 -9299.189} C_VEL
LIN {X 0,Y 432.311,Z 234.636,A -85,B 0,C 180,E1 -9302.444,E2 -9302.444} C_VEL
LIN {X 0,Y 432.334,Z 234.63,A -85,B 0,C 180,E1 -9305.634,E2 -9305.634} C_VEL
LIN {X 0,Y 432.35,Z 234.633,A -85,B 0,C 180,E1 -9308.72,E2 -9308.72} C_VEL
LIN {X 0,Y 432.364,Z 234.627,A -85,B 0,C 180,E1 -9311.794,E2 -9311.794} C_VEL
LIN {X 0,Y 432.369,Z 234.629,A -85,B 0,C 180,E1 -9314.343,E2 -9314.343} C_VEL
LIN {X 0,Y 432.357,Z 234.63,A -85,B 0,C 180,E1 -9317.011,E2 -9317.011} C_VEL
LIN {X 0,Y 432.35,Z 234.63,A -85,B 0,C 180,E1 -9319.819,E2 -9319.819} C_VEL
LIN {X 0,Y 432.31,Z 234.635,A -85,B 0,C 180,E1 -9323.025,E2 -9323.025} C_VEL
LIN {X 0,Y 432.353,Z 234.631,A -85,B 0,C 180,E1 -9325.998,E2 -9325.998} C_VEL
LIN {X 0,Y 432.39,Z 234.625,A -85,B 0,C 180,E1 -9329.746,E2 -9329.746} C_VEL
LIN {X 0,Y 432.396,Z 234.622,A -85,B 0,C 180,E1 -9333.374,E2 -9333.374} C_VEL
LIN {X 0,Y 432.368,Z 234.63,A -85,B 0,C 180,E1 -9336.025,E2 -9336.025} C_VEL
LIN {X 0,Y 432.348,Z 234.628,A -85,B 0,C 180,E1 -9339.048,E2 -9339.048} C_VEL
LIN {X 0,Y 432.377,Z 234.629,A -85,B 0,C 180,E1 -9342.013,E2 -9342.013} C_VEL
LIN {X 0,Y 432.394,Z 234.623,A -85,B 0,C 180,E1 -9344.928,E2 -9344.928} C_VEL
LIN {X 0,Y 432.459,Z 234.618,A -85,B 0,C 180,E1 -9347.805,E2 -9347.805} C_VEL
LIN {X 0,Y 432.464,Z 234.617,A -85,B 0,C 180,E1 -9351.591,E2 -9351.591} C_VEL
LIN {X 0,Y 432.597,Z 234.599,A -85,B 0,C 180,E1 -9354.408,E2 -9354.408} C_VEL
LIN {X 0,Y 432.605,Z 234.599,A -85,B 0,C 180,E1 -9358.14,E2 -9358.14} C_VEL
LIN {X 0,Y 432.735,Z 234.584,A -85,B 0,C 180,E1 -9360.002,E2 -9360.002} C_VEL
LIN {X 0,Y 432.593,Z 234.599,A -85,B 0,C 180,E1 -9362.795,E2 -9362.795} C_VEL
LIN {X 0,Y 432.588,Z 234.602,A -85,B 0,C 180,E1 -9365.595,E2 -9365.595} C_VEL
LIN {X 0,Y 432.468,Z 234.615,A -85,B 0,C 180,E1 -9368.412,E2 -9368.412} C_VEL
LIN {X 0,Y 432.464,Z 234.615,A -85,B 0,C 180,E1 -9372.198,E2 -9372.198} C_VEL
LIN {X 0,Y 432.436,Z 234.62,A -85,B 0,C 180,E1 -9376.04,E2 -9376.04} C_VEL
LIN {X 0,Y 432.393,Z 234.626,A -85,B 0,C 180,E1 -9379.486,E2 -9379.486} C_VEL
LIN {X 0,Y 432.322,Z 234.635,A -85,B 0,C 180,E1 -9382.965,E2 -9382.965} C_VEL
LIN {X 0,Y 432.356,Z 234.629,A -85,B 0,C 180,E1 -9386.034,E2 -9386.034} C_VEL
LIN {X 0,Y 432.349,Z 234.632,A -85,B 0,C 180,E1 -9389.188,E2 -9389.188} C_VEL
LIN {X 0,Y 432.328,Z 234.632,A -85,B 0,C 180,E1 -9392.444,E2 -9392.444} C_VEL
LIN {X 0,Y 432.349,Z 234.631,A -85,B 0,C 180,E1 -9395.632,E2 -9395.632} C_VEL
LIN {X 0,Y 432.346,Z 234.632,A -85,B 0,C 180,E1 -9398.715,E2 -9398.715} C_VEL
LIN {X 0,Y 432.34,Z 234.631,A -85,B 0,C 180,E1 -9401.798,E2 -9401.798} C_VEL
LIN {X 0,Y 432.34,Z 234.63,A -85,B 0,C 180,E1 -9404.348,E2 -9404.348} C_VEL
LIN {X 0,Y 432.395,Z 234.787,A -85,B 0,C 180,E1 -9407.503,E2 -9407.503} C_VEL
LIN {X 0,Y 433.405,Z 240.23,A -85,B 0,C 180,E1 -9410.241,E2 -9410.241} C_VEL
LIN {X 0,Y 434.414,Z 246.514,A -85,B 0,C 180,E1 -9413.231,E2 -9413.231} C_VEL
LIN {X 0,Y 434.389,Z 250.391,A -85,B 0,C 180,E1 -9414.945,E2 -9414.945} C_VEL
LIN {X 0,Y 433.94,Z 256.858,A -85,B 0,C 180,E1 -9417.692,E2 -9417.692} C_VEL
LIN {X 0,Y 433.392,Z 264.681,A -85,B 0,C 180,E1 -9420.89,E2 -9420.89} C_VEL
LIN {X 0,Y 432.957,Z 272.536,A -85,B 0,C 180,E1 -9424.005,E2 -9424.005} C_VEL
LIN {X 0,Y 432.554,Z 280.449,A -85,B 0,C 180,E1 -9427.049,E2 -9427.049} C_VEL
LIN {X 0,Y 432.179,Z 289.975,A -85,B 0,C 180,E1 -9430.595,E2 -9430.595} C_VEL
LIN {X 0,Y 431.87,Z 297.435,A -85,B 0,C 180,E1 -9433.296,E2 -9433.296} C_VEL
LIN {X 0,Y 434.066,Z 310.984,A -85,B 0,C 180,E1 -9433.763,E2 -9433.763} C_VEL
LIN {X 0,Y 435.64,Z 321.399,A -85,B 0,C 180,E1 -9434.262,E2 -9434.262} C_VEL
LIN {X 0,Y 435.089,Z 333.068,A -85,B 0,C 180,E1 -9434.902,E2 -9434.902} C_VEL
LIN {X 0,Y 434.449,Z 344.457,A -85,B 0,C 180,E1 -9435.717,E2 -9435.717} C_VEL
LIN {X 0,Y 433.828,Z 355.368,A -85,B 0,C 180,E1 -9436.703,E2 -9436.703} C_VEL
LIN {X 0,Y 433.208,Z 365.4,A -85,B 0,C 180,E1 -9437.824,E2 -9437.824} C_VEL
LIN {X 0,Y 432.561,Z 373.934,A -85,B 0,C 180,E1 -9438.994,E2 -9438.994} C_VEL
LIN {X 0,Y 432.106,Z 382.268,A -85,B 0,C 180,E1 -9440.403,E2 -9440.403} C_VEL
LIN {X 0,Y 431.714,Z 388.987,A -85,B 0,C 180,E1 -9441.81,E2 -9441.81} C_VEL
LIN {X 0,Y 431.452,Z 395.146,A -85,B 0,C 180,E1 -9443.452,E2 -9443.452} C_VEL
LIN {X 0,Y 431.35,Z 399.149,A -85,B 0,C 180,E1 -9444.858,E2 -9444.858} C_VEL
LIN {X 0,Y 431.21,Z 402.099,A -85,B 0,C 180,E1 -9446.262,E2 -9446.262} C_VEL
LIN {X 0,Y 431.281,Z 403.512,A -85,B 0,C 180,E1 -9447.197,E2 -9447.197} C_VEL
LIN {X 0,Y 431.185,Z 405.118,A -85,B 0,C 180,E1 -9449.066,E2 -9449.066} C_VEL
LIN {X 0,Y 431.204,Z 405.332,A -85,B 0,C 180,E1 -9449.999,E2 -9449.999} C_VEL
LIN {X 0,Y 431.185,Z 405.107,A -85,B 0,C 180,E1 -9450.933,E2 -9450.933} C_VEL
LIN {X 0,Y 431.281,Z 403.478,A -85,B 0,C 180,E1 -9452.802,E2 -9452.802} C_VEL
LIN {X 0,Y 431.211,Z 402.052,A -85,B 0,C 180,E1 -9453.737,E2 -9453.737} C_VEL
LIN {X 0,Y 431.37,Z 399.078,A -85,B 0,C 180,E1 -9455.14,E2 -9455.14} C_VEL
LIN {X 0,Y 431.444,Z 395.047,A -85,B 0,C 180,E1 -9456.547,E2 -9456.547} C_VEL
LIN {X 0,Y 431.713,Z 388.862,A -85,B 0,C 180,E1 -9458.189,E2 -9458.189} C_VEL
LIN {X 0,Y 432.083,Z 382.111,A -85,B 0,C 180,E1 -9459.597,E2 -9459.597} C_VEL
LIN {X 0,Y 432.56,Z 373.742,A -85,B 0,C 180,E1 -9461.005,E2 -9461.005} C_VEL
LIN {X 0,Y 433.201,Z 365.178,A -85,B 0,C 180,E1 -9462.175,E2 -9462.175} C_VEL
LIN {X 0,Y 433.782,Z 355.293,A -85,B 0,C 180,E1 -9463.279,E2 -9463.279} C_VEL
LIN {X 0,Y 434.375,Z 344.162,A -85,B 0,C 180,E1 -9464.284,E2 -9464.284} C_VEL
LIN {X 0,Y 435.065,Z 332.748,A -85,B 0,C 180,E1 -9465.098,E2 -9465.098} C_VEL
LIN {X 0,Y 435.539,Z 321.043,A -85,B 0,C 180,E1 -9465.741,E2 -9465.741} C_VEL
LIN {X 0,Y 433.477,Z 307.286,A -85,B 0,C 180,E1 -9466.369,E2 -9466.369} C_VEL
LIN {X 0,Y 431.839,Z 296.793,A -85,B 0,C 180,E1 -9466.72,E2 -9466.72} C_VEL
LIN {X 0,Y 432.187,Z 287.845,A -85,B 0,C 180,E1 -9469.967,E2 -9469.967} C_VEL
LIN {X 0,Y 432.488,Z 279.799,A -85,B 0,C 180,E1 -9472.954,E2 -9472.954} C_VEL
LIN {X 0,Y 432.851,Z 271.808,A -85,B 0,C 180,E1 -9476,E2 -9476} C_VEL
LIN {X 0,Y 433.342,Z 263.95,A -85,B 0,C 180,E1 -9479.113,E2 -9479.113} C_VEL
LIN {X 0,Y 433.831,Z 256.203,A -85,B 0,C 180,E1 -9482.316,E2 -9482.316} C_VEL
LIN {X 0,Y 434.462,Z 248.641,A -85,B 0,C 180,E1 -9485.615,E2 -9485.615} C_VEL
LIN {X 0,Y 434.145,Z 244.661,A -85,B 0,C 180,E1 -9487.511,E2 -9487.511} C_VEL
LIN {X 0,Y 432.948,Z 237.869,A -85,B 0,C 180,E1 -9491.061,E2 -9491.061} C_VEL
LIN {X 0,Y 432.322,Z 234.637,A -85,B 0,C 180,E1 -9492.983,E2 -9492.983} C_VEL
LIN {X 0,Y 432.335,Z 234.634,A -85,B 0,C 180,E1 -9495.664,E2 -9495.664} C_VEL
LIN {X 0,Y 432.368,Z 234.629,A -85,B 0,C 180,E1 -9498.392,E2 -9498.392} C_VEL
LIN {X 0,Y 432.353,Z 234.632,A -85,B 0,C 180,E1 -9501.85,E2 -9501.85} C_VEL
LIN {X 0,Y 432.34,Z 234.633,A -85,B 0,C 180,E1 -9505.322,E2 -9505.322} C_VEL
LIN {X 0,Y 432.321,Z 234.634,A -85,B 0,C 180,E1 -9508.653,E2 -9508.653} C_VEL
LIN {X 0,Y 432.383,Z 234.628,A -85,B 0,C 180,E1 -9511.875,E2 -9511.875} C_VEL
LIN {X 0,Y 432.351,Z 234.631,A -85,B 0,C 180,E1 -9514.997,E2 -9514.997} C_VEL
LIN {X 0,Y 432.357,Z 234.629,A -85,B 0,C 180,E1 -9518.044,E2 -9518.044} C_VEL
LIN {X 0,Y 432.385,Z 234.626,A -85,B 0,C 180,E1 -9521.028,E2 -9521.028} C_VEL
LIN {X 0,Y 432.429,Z 234.62,A -85,B 0,C 180,E1 -9523.96,E2 -9523.96} C_VEL
LIN {X 0,Y 432.457,Z 234.619,A -85,B 0,C 180,E1 -9527.802,E2 -9527.802} C_VEL
LIN {X 0,Y 432.489,Z 234.612,A -85,B 0,C 180,E1 -9531.589,E2 -9531.589} C_VEL
LIN {X 0,Y 432.595,Z 234.601,A -85,B 0,C 180,E1 -9534.405,E2 -9534.405} C_VEL
LIN {X 0,Y 432.602,Z 234.599,A -85,B 0,C 180,E1 -9538.137,E2 -9538.137} C_VEL
LIN {X 0,Y 432.731,Z 234.584,A -85,B 0,C 180,E1 -9539.998,E2 -9539.998} C_VEL
LIN {X 0,Y 432.6,Z 234.6,A -85,B 0,C 180,E1 -9542.792,E2 -9542.792} C_VEL
LIN {X 0,Y 432.567,Z 234.606,A -85,B 0,C 180,E1 -9546.529,E2 -9546.529} C_VEL
LIN {X 0,Y 432.431,Z 234.622,A -85,B 0,C 180,E1 -9549.352,E2 -9549.352} C_VEL
LIN {X 0,Y 432.221,Z 234.654,A -85,B 0,C 180,E1 -9552.683,E2 -9552.683} C_VEL
LIN {X 0,Y 432.062,Z 235.285,A -85,B 0,C 180,E1 -9554.12,E2 -9554.12} C_VEL
LIN {X 0,Y 431.985,Z 238.076,A -85,B 0,C 180,E1 -9557.026,E2 -9557.026} C_VEL
LIN {X 0,Y 431.884,Z 240.982,A -85,B 0,C 180,E1 -9559.98,E2 -9559.98} C_VEL
LIN {X 0,Y 431.78,Z 243.959,A -85,B 0,C 180,E1 -9562.992,E2 -9562.992} C_VEL
LIN {X 0,Y 431.708,Z 247.022,A -85,B 0,C 180,E1 -9566.073,E2 -9566.073} C_VEL
LIN {X 0,Y 431.611,Z 250.253,A -85,B 0,C 180,E1 -9569.239,E2 -9569.239} C_VEL
LIN {X 0,Y 431.613,Z 251.485,A -85,B 0,C 180,E1 -9570.415,E2 -9570.415} C_VEL
LIN {X 0,Y 435.091,Z 264.975,A -85,B 0,C 180,E1 -9571.021,E2 -9571.021} C_VEL
LIN {X 0,Y 436.178,Z 270.279,A -85,B 0,C 180,E1 -9571.305,E2 -9571.305} C_VEL
LIN {X 0,Y 435.686,Z 282.192,A -85,B 0,C 180,E1 -9571.955,E2 -9571.955} C_VEL
LIN {X 0,Y 435.096,Z 293.444,A -85,B 0,C 180,E1 -9572.761,E2 -9572.761} C_VEL
LIN {X 0,Y 434.416,Z 304.704,A -85,B 0,C 180,E1 -9573.785,E2 -9573.785} C_VEL
LIN {X 0,Y 433.772,Z 315.081,A -85,B 0,C 180,E1 -9574.968,E2 -9574.968} C_VEL
LIN {X 0,Y 433.146,Z 324.53,A -85,B 0,C 180,E1 -9576.322,E2 -9576.322} C_VEL
LIN {X 0,Y 432.601,Z 332.102,A -85,B 0,C 180,E1 -9577.662,E2 -9577.662} C_VEL
LIN {X 0,Y 432.176,Z 338.21,A -85,B 0,C 180,E1 -9578.998,E2 -9578.998} C_VEL
LIN {X 0,Y 431.819,Z 343.993,A -85,B 0,C 180,E1 -9580.615,E2 -9580.615} C_VEL
LIN {X 0,Y 431.556,Z 348.579,A -85,B 0,C 180,E1 -9582.37,E2 -9582.37} C_VEL
LIN {X 0,Y 431.444,Z 350.144,A -85,B 0,C 180,E1 -9583.166,E2 -9583.166} C_VEL
LIN {X 0,Y 431.288,Z 352.029,A -85,B 0,C 180,E1 -9584.48,E2 -9584.48} C_VEL
LIN {X 0,Y 431.228,Z 353.127,A -85,B 0,C 180,E1 -9585.812,E2 -9585.812} C_VEL
LIN {X 0,Y 431.209,Z 353.422,A -85,B 0,C 180,E1 -9587.171,E2 -9587.171} C_VEL
LIN {X 0,Y 431.206,Z 352.857,A -85,B 0,C 180,E1 -9588.564,E2 -9588.564} C_VEL
LIN {X 0,Y 431.323,Z 351.36,A -85,B 0,C 180,E1 -9589.976,E2 -9589.976} C_VEL
LIN {X 0,Y 431.505,Z 348.085,A -85,B 0,C 180,E1 -9591.764,E2 -9591.764} C_VEL
LIN {X 0,Y 431.676,Z 345.026,A -85,B 0,C 180,E1 -9592.96,E2 -9592.96} C_VEL
LIN {X 0,Y 431.979,Z 340.117,A -85,B 0,C 180,E1 -9594.432,E2 -9594.432} C_VEL
LIN {X 0,Y 432.357,Z 333.423,A -85,B 0,C 180,E1 -9595.993,E2 -9595.993} C_VEL
LIN {X 0,Y 432.859,Z 326.248,A -85,B 0,C 180,E1 -9597.328,E2 -9597.328} C_VEL
LIN {X 0,Y 433.464,Z 316.739,A -85,B 0,C 180,E1 -9598.747,E2 -9598.747} C_VEL
LIN {X 0,Y 434.086,Z 306.23,A -85,B 0,C 180,E1 -9600,E2 -9600} C_VEL
LIN {X 0,Y 434.725,Z 295.875,A -85,B 0,C 180,E1 -9600.989,E2 -9600.989} C_VEL
LIN {X 0,Y 435.278,Z 284.033,A -85,B 0,C 180,E1 -9601.885,E2 -9601.885} C_VEL
LIN {X 0,Y 435.847,Z 271.878,A -85,B 0,C 180,E1 -9602.59,E2 -9602.59} C_VEL
LIN {X 0,Y 435.731,Z 268.175,A -85,B 0,C 180,E1 -9602.773,E2 -9602.773} C_VEL
LIN {X 0,Y 432.815,Z 255.319,A -85,B 0,C 180,E1 -9603.387,E2 -9603.387} C_VEL
LIN {X 0,Y 431.549,Z 250.095,A -85,B 0,C 180,E1 -9603.594,E2 -9603.594} C_VEL
LIN {X 0,Y 431.53,Z 246.412,A -85,B 0,C 180,E1 -9606.992,E2 -9606.992} C_VEL
LIN {X 0,Y 431.644,Z 242.36,A -85,B 0,C 180,E1 -9610.788,E2 -9610.788} C_VEL
LIN {X 0,Y 431.73,Z 239.072,A -85,B 0,C 180,E1 -9613.935,E2 -9613.935} C_VEL
LIN {X 0,Y 431.842,Z 235.087,A -85,B 0,C 180,E1 -9617.786,E2 -9617.786} C_VEL
LIN {X 0,Y 432.039,Z 234.672,A -85,B 0,C 180,E1 -9619.693,E2 -9619.693} C_VEL
LIN {X 0,Y 432.336,Z 234.633,A -85,B 0,C 180,E1 -9621.719,E2 -9621.719} C_VEL
LIN {X 0,Y 431.741,Z 234.706,A -85,B 0,C 180,E1 -9622.498,E2 -9622.498} C_VEL
LIN {X 0,Y 428.912,Z 235.059,A -85,B 0,C 180,E1 -9623.765,E2 -9623.765} C_VEL
LIN {X 0,Y 426.47,Z 235.363,A -85,B 0,C 180,E1 -9624.787,E2 -9624.787} C_VEL
LIN {X 0,Y 425.413,Z 235.497,A -85,B 0,C 180,E1 -9625.578,E2 -9625.578} C_VEL
LIN {X 0,Y 425.324,Z 235.503,A -85,B 0,C 180,E1 -9625.845,E2 -9625.845} C_VEL
LIN {X 0,Y 425.56,Z 235.475,A -85,B 0,C 180,E1 -9628.108,E2 -9628.108} C_VEL
LIN {X 0,Y 425.688,Z 235.459,A -85,B 0,C 180,E1 -9630.001,E2 -9630.001} C_VEL
LIN {X 0,Y 425.543,Z 235.478,A -85,B 0,C 180,E1 -9632.84,E2 -9632.84} C_VEL
LIN {X 0,Y 425.516,Z 235.481,A -85,B 0,C 180,E1 -9636.64,E2 -9636.64} C_VEL
LIN {X 0,Y 425.389,Z 235.498,A -85,B 0,C 180,E1 -9639.51,E2 -9639.51} C_VEL
LIN {X 0,Y 425.388,Z 235.499,A -85,B 0,C 180,E1 -9642.911,E2 -9642.911} C_VEL
LIN {X 0,Y 425.346,Z 235.504,A -85,B 0,C 180,E1 -9646.606,E2 -9646.606} C_VEL
LIN {X 0,Y 425.348,Z 235.502,A -85,B 0,C 180,E1 -9649.65,E2 -9649.65} C_VEL
LIN {X 0,Y 425.291,Z 235.51,A -85,B 0,C 180,E1 -9652.339,E2 -9652.339} C_VEL
LIN {X 0,Y 425.287,Z 235.51,A -85,B 0,C 180,E1 -9655.446,E2 -9655.446} C_VEL
LIN {X 0,Y 425.318,Z 235.508,A -85,B 0,C 180,E1 -9658.634,E2 -9658.634} C_VEL
LIN {X 0,Y 425.253,Z 235.513,A -85,B 0,C 180,E1 -9661.928,E2 -9661.928} C_VEL
LIN {X 0,Y 425.289,Z 235.509,A -85,B 0,C 180,E1 -9665.337,E2 -9665.337} C_VEL
LIN {X 0,Y 425.303,Z 235.508,A -85,B 0,C 180,E1 -9669.048,E2 -9669.048} C_VEL
LIN {X 0,Y 425.322,Z 235.507,A -85,B 0,C 180,E1 -9672.648,E2 -9672.648} C_VEL
LIN {X 0,Y 425.325,Z 235.506,A -85,B 0,C 180,E1 -9676.055,E2 -9676.055} C_VEL
LIN {X 0,Y 425.302,Z 235.51,A -85,B 0,C 180,E1 -9678.627,E2 -9678.627} C_VEL
LIN {X 0,Y 425.317,Z 235.505,A -85,B 0,C 180,E1 -9681.106,E2 -9681.106} C_VEL
LIN {X 0,Y 425.294,Z 235.51,A -85,B 0,C 180,E1 -9684.666,E2 -9684.666} C_VEL
LIN {X 0,Y 425.267,Z 235.515,A -85,B 0,C 180,E1 -9688.076,E2 -9688.076} C_VEL
LIN {X 0,Y 425.333,Z 235.503,A -85,B 0,C 180,E1 -9691.37,E2 -9691.37} C_VEL
LIN {X 0,Y 425.292,Z 235.511,A -85,B 0,C 180,E1 -9694.557,E2 -9694.557} C_VEL
LIN {X 0,Y 425.285,Z 235.511,A -85,B 0,C 180,E1 -9697.663,E2 -9697.663} C_VEL
LIN {X 0,Y 425.36,Z 235.501,A -85,B 0,C 180,E1 -9700.706,E2 -9700.706} C_VEL
LIN {X 0,Y 425.387,Z 235.499,A -85,B 0,C 180,E1 -9703.69,E2 -9703.69} C_VEL
LIN {X 0,Y 425.412,Z 235.495,A -85,B 0,C 180,E1 -9707.6,E2 -9707.6} C_VEL
LIN {X 0,Y 425.409,Z 235.495,A -85,B 0,C 180,E1 -9711.451,E2 -9711.451} C_VEL
LIN {X 0,Y 425.552,Z 235.477,A -85,B 0,C 180,E1 -9714.315,E2 -9714.315} C_VEL
LIN {X 0,Y 425.575,Z 235.475,A -85,B 0,C 180,E1 -9718.109,E2 -9718.109} C_VEL
LIN {X 0,Y 425.704,Z 235.46,A -85,B 0,C 180,E1 -9720.002,E2 -9720.002} C_VEL
LIN {X 0,Y 425.547,Z 235.476,A -85,B 0,C 180,E1 -9722.841,E2 -9722.841} C_VEL
LIN {X 0,Y 425.544,Z 235.48,A -85,B 0,C 180,E1 -9725.688,E2 -9725.688} C_VEL
LIN {X 0,Y 425.412,Z 235.493,A -85,B 0,C 180,E1 -9728.552,E2 -9728.552} C_VEL
LIN {X 0,Y 425.417,Z 235.492,A -85,B 0,C 180,E1 -9732.403,E2 -9732.403} C_VEL
LIN {X 0,Y 425.394,Z 235.496,A -85,B 0,C 180,E1 -9736.313,E2 -9736.313} C_VEL
LIN {X 0,Y 425.334,Z 235.505,A -85,B 0,C 180,E1 -9739.637,E2 -9739.637} C_VEL
LIN {X 0,Y 425.309,Z 235.509,A -85,B 0,C 180,E1 -9743.366,E2 -9743.366} C_VEL
LIN {X 0,Y 425.346,Z 235.503,A -85,B 0,C 180,E1 -9746.843,E2 -9746.843} C_VEL
LIN {X 0,Y 425.297,Z 235.509,A -85,B 0,C 180,E1 -9749.72,E2 -9749.72} C_VEL
LIN {X 0,Y 425.288,Z 235.511,A -85,B 0,C 180,E1 -9753.049,E2 -9753.049} C_VEL
LIN {X 0,Y 425.288,Z 235.509,A -85,B 0,C 180,E1 -9755.929,E2 -9755.929} C_VEL
LIN {X 0,Y 425.289,Z 235.511,A -85,B 0,C 180,E1 -9759.041,E2 -9759.041} C_VEL
LIN {X 0,Y 425.296,Z 235.508,A -85,B 0,C 180,E1 -9761.959,E2 -9761.959} C_VEL
LIN {X 0,Y 425.291,Z 235.508,A -85,B 0,C 180,E1 -9765.284,E2 -9765.284} C_VEL
LIN {X 0,Y 425.322,Z 235.635,A -85,B 0,C 180,E1 -9767.144,E2 -9767.144} C_VEL
LIN {X 0,Y 426.372,Z 241.16,A -85,B 0,C 180,E1 -9769.995,E2 -9769.995} C_VEL
LIN {X 0,Y 427.404,Z 247.618,A -85,B 0,C 180,E1 -9773.117,E2 -9773.117} C_VEL
LIN {X 0,Y 427.418,Z 251.471,A -85,B 0,C 180,E1 -9774.865,E2 -9774.865} C_VEL
LIN {X 0,Y 426.864,Z 259.246,A -85,B 0,C 180,E1 -9778.206,E2 -9778.206} C_VEL
LIN {X 0,Y 426.25,Z 268.367,A -85,B 0,C 180,E1 -9781.971,E2 -9781.971} C_VEL
LIN {X 0,Y 425.695,Z 277.534,A -85,B 0,C 180,E1 -9785.623,E2 -9785.623} C_VEL
LIN {X 0,Y 425.283,Z 285.421,A -85,B 0,C 180,E1 -9788.681,E2 -9788.681} C_VEL
LIN {X 0,Y 424.951,Z 293.379,A -85,B 0,C 180,E1 -9791.685,E2 -9791.685} C_VEL
LIN {X 0,Y 424.802,Z 296.885,A -85,B 0,C 180,E1 -9792.992,E2 -9792.992} C_VEL
LIN {X 0,Y 427.145,Z 311.648,A -85,B 0,C 180,E1 -9793.534,E2 -9793.534} C_VEL
LIN {X 0,Y 428.7,Z 323.34,A -85,B 0,C 180,E1 -9794.123,E2 -9794.123} C_VEL
LIN {X 0,Y 427.981,Z 336.173,A -85,B 0,C 180,E1 -9794.889,E2 -9794.889} C_VEL
LIN {X 0,Y 427.331,Z 346.882,A -85,B 0,C 180,E1 -9795.718,E2 -9795.718} C_VEL
LIN {X 0,Y 426.677,Z 357.848,A -85,B 0,C 180,E1 -9796.788,E2 -9796.788} C_VEL
LIN {X 0,Y 426.098,Z 366.79,A -85,B 0,C 180,E1 -9797.86,E2 -9797.86} C_VEL
LIN {X 0,Y 425.376,Z 376.506,A -85,B 0,C 180,E1 -9799.288,E2 -9799.288} C_VEL
LIN {X 0,Y 424.905,Z 384.263,A -85,B 0,C 180,E1 -9800.719,E2 -9800.719} C_VEL
LIN {X 0,Y 424.469,Z 391.406,A -85,B 0,C 180,E1 -9802.388,E2 -9802.388} C_VEL
LIN {X 0,Y 424.278,Z 396.556,A -85,B 0,C 180,E1 -9803.948,E2 -9803.948} C_VEL
LIN {X 0,Y 424.225,Z 399.808,A -85,B 0,C 180,E1 -9805.248,E2 -9805.248} C_VEL
LIN {X 0,Y 424.12,Z 401.681,A -85,B 0,C 180,E1 -9806.199,E2 -9806.199} C_VEL
LIN {X 0,Y 424.193,Z 403.094,A -85,B 0,C 180,E1 -9807.151,E2 -9807.151} C_VEL
LIN {X 0,Y 424.104,Z 404.698,A -85,B 0,C 180,E1 -9809.05,E2 -9809.05} C_VEL
LIN {X 0,Y 424.119,Z 404.911,A -85,B 0,C 180,E1 -9809.999,E2 -9809.999} C_VEL
LIN {X 0,Y 424.104,Z 404.685,A -85,B 0,C 180,E1 -9810.949,E2 -9810.949} C_VEL
LIN {X 0,Y 424.193,Z 403.049,A -85,B 0,C 180,E1 -9812.848,E2 -9812.848} C_VEL
LIN {X 0,Y 424.122,Z 401.62,A -85,B 0,C 180,E1 -9813.8,E2 -9813.8} C_VEL
LIN {X 0,Y 424.281,Z 398.642,A -85,B 0,C 180,E1 -9815.227,E2 -9815.227} C_VEL
LIN {X 0,Y 424.363,Z 394.605,A -85,B 0,C 180,E1 -9816.657,E2 -9816.657} C_VEL
LIN {X 0,Y 424.653,Z 388.412,A -85,B 0,C 180,E1 -9818.326,E2 -9818.326} C_VEL
LIN {X 0,Y 425.032,Z 381.653,A -85,B 0,C 180,E1 -9819.757,E2 -9819.757} C_VEL
LIN {X 0,Y 425.557,Z 373.279,A -85,B 0,C 180,E1 -9821.189,E2 -9821.189} C_VEL
LIN {X 0,Y 426.2,Z 364.707,A -85,B 0,C 180,E1 -9822.378,E2 -9822.378} C_VEL
LIN {X 0,Y 426.848,Z 354.174,A -85,B 0,C 180,E1 -9823.564,E2 -9823.564} C_VEL
LIN {X 0,Y 427.549,Z 342.247,A -85,B 0,C 180,E1 -9824.639,E2 -9824.639} C_VEL
LIN {X 0,Y 428.322,Z 330.328,A -85,B 0,C 180,E1 -9825.463,E2 -9825.463} C_VEL
LIN {X 0,Y 428.619,Z 321.8,A -85,B 0,C 180,E1 -9825.94,E2 -9825.94} C_VEL
LIN {X 0,Y 426.682,Z 308.57,A -85,B 0,C 180,E1 -9826.579,E2 -9826.579} C_VEL
LIN {X 0,Y 424.773,Z 296.326,A -85,B 0,C 180,E1 -9827.008,E2 -9827.008} C_VEL
LIN {X 0,Y 425.109,Z 288.618,A -85,B 0,C 180,E1 -9829.873,E2 -9829.873} C_VEL
LIN {X 0,Y 425.458,Z 279.44,A -85,B 0,C 180,E1 -9833.356,E2 -9833.356} C_VEL
LIN {X 0,Y 425.884,Z 271.473,A -85,B 0,C 180,E1 -9836.458,E2 -9836.458} C_VEL
LIN {X 0,Y 426.367,Z 263.631,A -85,B 0,C 180,E1 -9839.636,E2 -9839.636} C_VEL
LIN {X 0,Y 426.921,Z 255.975,A -85,B 0,C 180,E1 -9842.904,E2 -9842.904} C_VEL
LIN {X 0,Y 427.496,Z 249.772,A -85,B 0,C 180,E1 -9845.704,E2 -9845.704} C_VEL
LIN {X 0,Y 427.185,Z 246.072,A -85,B 0,C 180,E1 -9847.496,E2 -9847.496} C_VEL
LIN {X 0,Y 426.153,Z 240.119,A -85,B 0,C 180,E1 -9850.656,E2 -9850.656} C_VEL
LIN {X 0,Y 425.274,Z 235.517,A -85,B 0,C 180,E1 -9853.352,E2 -9853.352} C_VEL
LIN {X 0,Y 425.259,Z 235.516,A -85,B 0,C 180,E1 -9856.648,E2 -9856.648} C_VEL
LIN {X 0,Y 425.301,Z 235.511,A -85,B 0,C 180,E1 -9859.475,E2 -9859.475} C_VEL
LIN {X 0,Y 425.287,Z 235.513,A -85,B 0,C 180,E1 -9862.486,E2 -9862.486} C_VEL
LIN {X 0,Y 425.307,Z 235.51,A -85,B 0,C 180,E1 -9865.816,E2 -9865.816} C_VEL
LIN {X 0,Y 425.29,Z 235.511,A -85,B 0,C 180,E1 -9869.238,E2 -9869.238} C_VEL
LIN {X 0,Y 425.35,Z 235.504,A -85,B 0,C 180,E1 -9872.441,E2 -9872.441} C_VEL
LIN {X 0,Y 425.351,Z 235.503,A -85,B 0,C 180,E1 -9875.601,E2 -9875.601} C_VEL
LIN {X 0,Y 425.293,Z 235.51,A -85,B 0,C 180,E1 -9878.68,E2 -9878.68} C_VEL
LIN {X 0,Y 425.332,Z 235.504,A -85,B 0,C 180,E1 -9881.701,E2 -9881.701} C_VEL
LIN {X 0,Y 425.346,Z 235.502,A -85,B 0,C 180,E1 -9884.669,E2 -9884.669} C_VEL
LIN {X 0,Y 425.409,Z 235.496,A -85,B 0,C 180,E1 -9887.597,E2 -9887.597} C_VEL
LIN {X 0,Y 425.439,Z 235.49,A -85,B 0,C 180,E1 -9891.448,E2 -9891.448} C_VEL
LIN {X 0,Y 425.552,Z 235.479,A -85,B 0,C 180,E1 -9894.312,E2 -9894.312} C_VEL
LIN {X 0,Y 425.572,Z 235.475,A -85,B 0,C 180,E1 -9898.106,E2 -9898.106} C_VEL
LIN {X 0,Y 425.7,Z 235.459,A -85,B 0,C 180,E1 -9899.998,E2 -9899.998} C_VEL
LIN {X 0,Y 425.552,Z 235.478,A -85,B 0,C 180,E1 -9902.838,E2 -9902.838} C_VEL
LIN {X 0,Y 425.525,Z 235.483,A -85,B 0,C 180,E1 -9906.644,E2 -9906.644} C_VEL
LIN {X 0,Y 425.387,Z 235.5,A -85,B 0,C 180,E1 -9909.508,E2 -9909.508} C_VEL
LIN {X 0,Y 425.18,Z 235.531,A -85,B 0,C 180,E1 -9912.78,E2 -9912.78} C_VEL
LIN {X 0,Y 425.046,Z 235.569,A -85,B 0,C 180,E1 -9913.383,E2 -9913.383} C_VEL
LIN {X 0,Y 424.982,Z 238.418,A -85,B 0,C 180,E1 -9916.435,E2 -9916.435} C_VEL
LIN {X 0,Y 424.866,Z 241.325,A -85,B 0,C 180,E1 -9919.462,E2 -9919.462} C_VEL
LIN {X 0,Y 424.736,Z 244.194,A -85,B 0,C 180,E1 -9922.367,E2 -9922.367} C_VEL
LIN {X 0,Y 424.651,Z 247.261,A -85,B 0,C 180,E1 -9925.485,E2 -9925.485} C_VEL
LIN {X 0,Y 424.586,Z 250.458,A -85,B 0,C 180,E1 -9928.685,E2 -9928.685} C_VEL
LIN {X 0,Y 424.549,Z 251.908,A -85,B 0,C 180,E1 -9930.106,E2 -9930.106} C_VEL
LIN {X 0,Y 428.191,Z 265.884,A -85,B 0,C 180,E1 -9930.766,E2 -9930.766} C_VEL
LIN {X 0,Y 429.363,Z 271.33,A -85,B 0,C 180,E1 -9931.07,E2 -9931.07} C_VEL
LIN {X 0,Y 428.816,Z 283.647,A -85,B 0,C 180,E1 -9931.767,E2 -9931.767} C_VEL
LIN {X 0,Y 428.131,Z 295.543,A -85,B 0,C 180,E1 -9932.658,E2 -9932.658} C_VEL
LIN {X 0,Y 427.434,Z 306.975,A -85,B 0,C 180,E1 -9933.749,E2 -9933.749} C_VEL
LIN {X 0,Y 426.79,Z 316.284,A -85,B 0,C 180,E1 -9934.862,E2 -9934.862} C_VEL
LIN {X 0,Y 426.148,Z 325.494,A -85,B 0,C 180,E1 -9936.22,E2 -9936.22} C_VEL
LIN {X 0,Y 425.552,Z 333.38,A -85,B 0,C 180,E1 -9937.663,E2 -9937.663} C_VEL
LIN {X 0,Y 425.052,Z 340.158,A -85,B 0,C 180,E1 -9939.247,E2 -9939.247} C_VEL
LIN {X 0,Y 424.709,Z 345.632,A -85,B 0,C 180,E1 -9940.909,E2 -9940.909} C_VEL
LIN {X 0,Y 424.563,Z 348.064,A -85,B 0,C 180,E1 -9941.85,E2 -9941.85} C_VEL
LIN {X 0,Y 424.364,Z 350.815,A -85,B 0,C 180,E1 -9943.224,E2 -9943.224} C_VEL
LIN {X 0,Y 424.21,Z 352.626,A -85,B 0,C 180,E1 -9944.571,E2 -9944.571} C_VEL
LIN {X 0,Y 424.137,Z 353.615,A -85,B 0,C 180,E1 -9945.898,E2 -9945.898} C_VEL
LIN {X 0,Y 424.121,Z 353.847,A -85,B 0,C 180,E1 -9947.204,E2 -9947.204} C_VEL
LIN {X 0,Y 424.131,Z 353.35,A -85,B 0,C 180,E1 -9948.486,E2 -9948.486} C_VEL
LIN {X 0,Y 424.228,Z 352.107,A -85,B 0,C 180,E1 -9949.753,E2 -9949.753} C_VEL
LIN {X 0,Y 424.422,Z 348.875,A -85,B 0,C 180,E1 -9951.67,E2 -9951.67} C_VEL
LIN {X 0,Y 424.694,Z 344.278,A -85,B 0,C 180,E1 -9953.435,E2 -9953.435} C_VEL
LIN {X 0,Y 425.042,Z 339.062,A -85,B 0,C 180,E1 -9954.929,E2 -9954.929} C_VEL
LIN {X 0,Y 425.435,Z 332.549,A -85,B 0,C 180,E1 -9956.4,E2 -9956.4} C_VEL
LIN {X 0,Y 425.966,Z 325.162,A -85,B 0,C 180,E1 -9957.736,E2 -9957.736} C_VEL
LIN {X 0,Y 426.639,Z 315.635,A -85,B 0,C 180,E1 -9959.128,E2 -9959.128} C_VEL
LIN {X 0,Y 427.213,Z 305.794,A -85,B 0,C 180,E1 -9960.293,E2 -9960.293} C_VEL
LIN {X 0,Y 427.901,Z 295.269,A -85,B 0,C 180,E1 -9961.288,E2 -9961.288} C_VEL
LIN {X 0,Y 428.502,Z 283.251,A -85,B 0,C 180,E1 -9962.194,E2 -9962.194} C_VEL
LIN {X 0,Y 429.066,Z 270.636,A -85,B 0,C 180,E1 -9962.913,E2 -9962.913} C_VEL
LIN {X 0,Y 426.312,Z 257.826,A -85,B 0,C 180,E1 -9963.557,E2 -9963.557} C_VEL
LIN {X 0,Y 424.49,Z 250.46,A -85,B 0,C 180,E1 -9963.878,E2 -9963.878} C_VEL
LIN {X 0,Y 424.469,Z 246.464,A -85,B 0,C 180,E1 -9967.617,E2 -9967.617} C_VEL
LIN {X 0,Y 424.563,Z 243.221,A -85,B 0,C 180,E1 -9970.667,E2 -9970.667} C_VEL
LIN {X 0,Y 424.628,Z 240.036,A -85,B 0,C 180,E1 -9973.722,E2 -9973.722} C_VEL
LIN {X 0,Y 424.783,Z 236.077,A -85,B 0,C 180,E1 -9977.58,E2 -9977.58} C_VEL
LIN {X 0,Y 424.837,Z 235.569,A -85,B 0,C 180,E1 -9978.551,E2 -9978.551} C_VEL
LIN {X 0,Y 425.291,Z 235.509,A -85,B 0,C 180,E1 -9981.738,E2 -9981.738} C_VEL
LIN {X 0,Y 425.536,Z 235.478,A -85,B 0,C 180,E1 -9984.314,E2 -9984.314} C_VEL
LIN {X 0,Y 425.324,Z 235.503,A -85,B 0,C 180,E1 -9985.845,E2 -9985.845} C_VEL
LIN {X 0,Y 424.715,Z 235.581,A -85,B 0,C 180,E1 -9986.636,E2 -9986.636} C_VEL
LIN {X 0,Y 422.102,Z 235.907,A -85,B 0,C 180,E1 -9987.926,E2 -9987.926} C_VEL
LIN {X 0,Y 419.032,Z 236.291,A -85,B 0,C 180,E1 -9989.497,E2 -9989.497} C_VEL
LIN {X 0,Y 418.65,Z 236.335,A -85,B 0,C 180,E1 -9990.037,E2 -9990.037} C_VEL
LIN {X 0,Y 418.497,Z 236.356,A -85,B 0,C 180,E1 -9992.888,E2 -9992.888} C_VEL
LIN {X 0,Y 418.479,Z 236.359,A -85,B 0,C 180,E1 -9996.752,E2 -9996.752} C_VEL
LIN {X 0,Y 418.345,Z 236.375,A -85,B 0,C 180,E1 -9999.672,E2 -9999.672} C_VEL
LIN {X 0,Y 418.34,Z 236.377,A -85,B 0,C 180,E1 -10003.007,E2 -10003.007} C_VEL
LIN {X 0,Y 418.298,Z 236.382,A -85,B 0,C 180,E1 -10006.737,E2 -10006.737} C_VEL
LIN {X 0,Y 418.29,Z 236.38,A -85,B 0,C 180,E1 -10009.804,E2 -10009.804} C_VEL
LIN {X 0,Y 418.262,Z 236.386,A -85,B 0,C 180,E1 -10012.735,E2 -10012.735} C_VEL
LIN {X 0,Y 418.26,Z 236.384,A -85,B 0,C 180,E1 -10015.905,E2 -10015.905} C_VEL
LIN {X 0,Y 418.252,Z 236.387,A -85,B 0,C 180,E1 -10019.163,E2 -10019.163} C_VEL
LIN {X 0,Y 418.245,Z 236.389,A -85,B 0,C 180,E1 -10022.846,E2 -10022.846} C_VEL
LIN {X 0,Y 418.237,Z 236.388,A -85,B 0,C 180,E1 -10026.24,E2 -10026.24} C_VEL
LIN {X 0,Y 418.256,Z 236.384,A -85,B 0,C 180,E1 -10029.682,E2 -10029.682} C_VEL
LIN {X 0,Y 418.275,Z 236.385,A -85,B 0,C 180,E1 -10032.331,E2 -10032.331} C_VEL
LIN {X 0,Y 418.265,Z 236.384,A -85,B 0,C 180,E1 -10035.116,E2 -10035.116} C_VEL
LIN {X 0,Y 418.284,Z 236.381,A -85,B 0,C 180,E1 -10037.775,E2 -10037.775} C_VEL
LIN {X 0,Y 418.259,Z 236.383,A -85,B 0,C 180,E1 -10041.562,E2 -10041.562} C_VEL
LIN {X 0,Y 418.253,Z 236.385,A -85,B 0,C 180,E1 -10045.161,E2 -10045.161} C_VEL
LIN {X 0,Y 418.243,Z 236.385,A -85,B 0,C 180,E1 -10047.474,E2 -10047.474} C_VEL
LIN {X 0,Y 418.272,Z 236.383,A -85,B 0,C 180,E1 -10050.895,E2 -10050.895} C_VEL
LIN {X 0,Y 418.267,Z 236.387,A -85,B 0,C 180,E1 -10054.098,E2 -10054.098} C_VEL
LIN {X 0,Y 418.235,Z 236.387,A -85,B 0,C 180,E1 -10057.266,E2 -10057.266} C_VEL
LIN {X 0,Y 418.281,Z 236.384,A -85,B 0,C 180,E1 -10060.366,E2 -10060.366} C_VEL
LIN {X 0,Y 418.316,Z 236.378,A -85,B 0,C 180,E1 -10063.407,E2 -10063.407} C_VEL
LIN {X 0,Y 418.346,Z 236.373,A -85,B 0,C 180,E1 -10067.001,E2 -10067.001} C_VEL
LIN {X 0,Y 418.339,Z 236.376,A -85,B 0,C 180,E1 -10070.33,E2 -10070.33} C_VEL
LIN {X 0,Y 418.476,Z 236.358,A -85,B 0,C 180,E1 -10073.25,E2 -10073.25} C_VEL
LIN {X 0,Y 418.34,Z 236.374,A -85,B 0,C 180,E1 -10075.183,E2 -10075.183} C_VEL
LIN {X 0,Y 418.544,Z 236.351,A -85,B 0,C 180,E1 -10078.077,E2 -10078.077} C_VEL
LIN {X 0,Y 418.673,Z 236.335,A -85,B 0,C 180,E1 -10080.002,E2 -10080.002} C_VEL
LIN {X 0,Y 418.502,Z 236.354,A -85,B 0,C 180,E1 -10082.889,E2 -10082.889} C_VEL
LIN {X 0,Y 418.501,Z 236.358,A -85,B 0,C 180,E1 -10085.784,E2 -10085.784} C_VEL
LIN {X 0,Y 418.381,Z 236.369,A -85,B 0,C 180,E1 -10088.697,E2 -10088.697} C_VEL
LIN {X 0,Y 418.319,Z 236.38,A -85,B 0,C 180,E1 -10091.632,E2 -10091.632} C_VEL
LIN {X 0,Y 418.308,Z 236.378,A -85,B 0,C 180,E1 -10094.598,E2 -10094.598} C_VEL
LIN {X 0,Y 418.294,Z 236.383,A -85,B 0,C 180,E1 -10097.605,E2 -10097.605} C_VEL
LIN {X 0,Y 418.256,Z 236.385,A -85,B 0,C 180,E1 -10100.664,E2 -10100.664} C_VEL
LIN {X 0,Y 418.29,Z 236.382,A -85,B 0,C 180,E1 -10103.782,E2 -10103.782} C_VEL
LIN {X 0,Y 418.317,Z 236.379,A -85,B 0,C 180,E1 -10107.071,E2 -10107.071} C_VEL
LIN {X 0,Y 418.251,Z 236.385,A -85,B 0,C 180,E1 -10110.273,E2 -10110.273} C_VEL
LIN {X 0,Y 418.254,Z 236.386,A -85,B 0,C 180,E1 -10113.678,E2 -10113.678} C_VEL
LIN {X 0,Y 418.246,Z 236.389,A -85,B 0,C 180,E1 -10117.225,E2 -10117.225} C_VEL
LIN {X 0,Y 418.251,Z 236.385,A -85,B 0,C 180,E1 -10119.683,E2 -10119.683} C_VEL
LIN {X 0,Y 418.236,Z 236.387,A -85,B 0,C 180,E1 -10122.322,E2 -10122.322} C_VEL
LIN {X 0,Y 418.242,Z 236.386,A -85,B 0,C 180,E1 -10125.109,E2 -10125.109} C_VEL
LIN {X 0,Y 418.266,Z 236.591,A -85,B 0,C 180,E1 -10126.852,E2 -10126.852} C_VEL
LIN {X 0,Y 419.35,Z 242.231,A -85,B 0,C 180,E1 -10129.817,E2 -10129.817} C_VEL
LIN {X 0,Y 420.387,Z 248.677,A -85,B 0,C 180,E1 -10132.997,E2 -10132.997} C_VEL
LIN {X 0,Y 420.419,Z 253.015,A -85,B 0,C 180,E1 -10134.998,E2 -10134.998} C_VEL
LIN {X 0,Y 419.752,Z 261.383,A -85,B 0,C 180,E1 -10138.64,E2 -10138.64} C_VEL
LIN {X 0,Y 419.213,Z 269.393,A -85,B 0,C 180,E1 -10142.003,E2 -10142.003} C_VEL
LIN {X 0,Y 418.675,Z 277.233,A -85,B 0,C 180,E1 -10145.187,E2 -10145.187} C_VEL
LIN {X 0,Y 418.283,Z 285.113,A -85,B 0,C 180,E1 -10148.306,E2 -10148.306} C_VEL
LIN {X 0,Y 417.928,Z 293.002,A -85,B 0,C 180,E1 -10151.366,E2 -10151.366} C_VEL
LIN {X 0,Y 417.761,Z 296.458,A -85,B 0,C 180,E1 -10152.688,E2 -10152.688} C_VEL
LIN {X 0,Y 420.239,Z 312.129,A -85,B 0,C 180,E1 -10153.294,E2 -10153.294} C_VEL
LIN {X 0,Y 421.808,Z 324.039,A -85,B 0,C 180,E1 -10153.918,E2 -10153.918} C_VEL
LIN {X 0,Y 421.111,Z 335.75,A -85,B 0,C 180,E1 -10154.636,E2 -10154.636} C_VEL
LIN {X 0,Y 420.446,Z 346.459,A -85,B 0,C 180,E1 -10155.479,E2 -10155.479} C_VEL
LIN {X 0,Y 419.746,Z 357.424,A -85,B 0,C 180,E1 -10156.566,E2 -10156.566} C_VEL
LIN {X 0,Y 419.126,Z 366.367,A -85,B 0,C 180,E1 -10157.655,E2 -10157.655} C_VEL
LIN {X 0,Y 418.365,Z 376.084,A -85,B 0,C 180,E1 -10159.106,E2 -10159.106} C_VEL
LIN {X 0,Y 417.864,Z 383.843,A -85,B 0,C 180,E1 -10160.561,E2 -10160.561} C_VEL
LIN {X 0,Y 417.543,Z 389.155,A -85,B 0,C 180,E1 -10161.774,E2 -10161.774} C_VEL
LIN {X 0,Y 417.275,Z 394.308,A -85,B 0,C 180,E1 -10163.229,E2 -10163.229} C_VEL
LIN {X 0,Y 417.183,Z 398.313,A -85,B 0,C 180,E1 -10164.683,E2 -10164.683} C_VEL
LIN {X 0,Y 417.035,Z 401.263,A -85,B 0,C 180,E1 -10166.134,E2 -10166.134} C_VEL
LIN {X 0,Y 417.093,Z 402.675,A -85,B 0,C 180,E1 -10167.102,E2 -10167.102} C_VEL
LIN {X 0,Y 417.059,Z 403.674,A -85,B 0,C 180,E1 -10168.068,E2 -10168.068} C_VEL
LIN {X 0,Y 417.037,Z 404.49,A -85,B 0,C 180,E1 -10169.999,E2 -10169.999} C_VEL
LIN {X 0,Y 417.025,Z 404.262,A -85,B 0,C 180,E1 -10170.965,E2 -10170.965} C_VEL
LIN {X 0,Y 417.059,Z 403.638,A -85,B 0,C 180,E1 -10171.931,E2 -10171.931} C_VEL
LIN {X 0,Y 417.108,Z 402.62,A -85,B 0,C 180,E1 -10172.897,E2 -10172.897} C_VEL
LIN {X 0,Y 417.037,Z 401.189,A -85,B 0,C 180,E1 -10173.865,E2 -10173.865} C_VEL
LIN {X 0,Y 417.194,Z 398.205,A -85,B 0,C 180,E1 -10175.316,E2 -10175.316} C_VEL
LIN {X 0,Y 417.279,Z 394.162,A -85,B 0,C 180,E1 -10176.77,E2 -10176.77} C_VEL
LIN {X 0,Y 417.591,Z 387.961,A -85,B 0,C 180,E1 -10178.468,E2 -10178.468} C_VEL
LIN {X 0,Y 418.005,Z 381.196,A -85,B 0,C 180,E1 -10179.923,E2 -10179.923} C_VEL
LIN {X 0,Y 418.569,Z 372.819,A -85,B 0,C 180,E1 -10181.378,E2 -10181.378} C_VEL
LIN {X 0,Y 419.206,Z 364.241,A -85,B 0,C 180,E1 -10182.588,E2 -10182.588} C_VEL
LIN {X 0,Y 419.894,Z 353.515,A -85,B 0,C 180,E1 -10183.813,E2 -10183.813} C_VEL
LIN {X 0,Y 420.658,Z 341.789,A -85,B 0,C 180,E1 -10184.884,E2 -10184.884} C_VEL
LIN {X 0,Y 421.485,Z 329.88,A -85,B 0,C 180,E1 -10185.721,E2 -10185.721} C_VEL
LIN {X 0,Y 421.674,Z 322.483,A -85,B 0,C 180,E1 -10186.148,E2 -10186.148} C_VEL
LIN {X 0,Y 419.735,Z 308.871,A -85,B 0,C 180,E1 -10186.837,E2 -10186.837} C_VEL
LIN {X 0,Y 417.72,Z 295.876,A -85,B 0,C 180,E1 -10187.315,E2 -10187.315} C_VEL
LIN {X 0,Y 418.046,Z 288.385,A -85,B 0,C 180,E1 -10190.158,E2 -10190.158} C_VEL
LIN {X 0,Y 418.448,Z 279.086,A -85,B 0,C 180,E1 -10193.771,E2 -10193.771} C_VEL
LIN {X 0,Y 418.945,Z 270.467,A -85,B 0,C 180,E1 -10197.238,E2 -10197.238} C_VEL
LIN {X 0,Y 419.415,Z 263.44,A -85,B 0,C 180,E1 -10200.178,E2 -10200.178} C_VEL
LIN {X 0,Y 420.048,Z 255.83,A -85,B 0,C 180,E1 -10203.513,E2 -10203.513} C_VEL
LIN {X 0,Y 420.51,Z 250.883,A -85,B 0,C 180,E1 -10205.799,E2 -10205.799} C_VEL
LIN {X 0,Y 420.203,Z 247.316,A -85,B 0,C 180,E1 -10207.57,E2 -10207.57} C_VEL
LIN {X 0,Y 419.121,Z 240.99,A -85,B 0,C 180,E1 -10211.01,E2 -10211.01} C_VEL
LIN {X 0,Y 418.216,Z 236.394,A -85,B 0,C 180,E1 -10213.805,E2 -10213.805} C_VEL
LIN {X 0,Y 418.211,Z 236.393,A -85,B 0,C 180,E1 -10216.447,E2 -10216.447} C_VEL
LIN {X 0,Y 418.267,Z 236.387,A -85,B 0,C 180,E1 -10219.122,E2 -10219.122} C_VEL
LIN {X 0,Y 418.239,Z 236.391,A -85,B 0,C 180,E1 -10222.164,E2 -10222.164} C_VEL
LIN {X 0,Y 418.266,Z 236.386,A -85,B 0,C 180,E1 -10225.418,E2 -10225.418} C_VEL
LIN {X 0,Y 418.211,Z 236.392,A -85,B 0,C 180,E1 -10228.603,E2 -10228.603} C_VEL
LIN {X 0,Y 418.292,Z 236.383,A -85,B 0,C 180,E1 -10231.935,E2 -10231.935} C_VEL
LIN {X 0,Y 418.289,Z 236.383,A -85,B 0,C 180,E1 -10235.161,E2 -10235.161} C_VEL
LIN {X 0,Y 418.233,Z 236.389,A -85,B 0,C 180,E1 -10238.302,E2 -10238.302} C_VEL
LIN {X 0,Y 418.283,Z 236.384,A -85,B 0,C 180,E1 -10241.382,E2 -10241.382} C_VEL
LIN {X 0,Y 418.3,Z 236.379,A -85,B 0,C 180,E1 -10244.404,E2 -10244.404} C_VEL
LIN {X 0,Y 418.353,Z 236.374,A -85,B 0,C 180,E1 -10247.384,E2 -10247.384} C_VEL
LIN {X 0,Y 418.338,Z 236.377,A -85,B 0,C 180,E1 -10250.327,E2 -10250.327} C_VEL
LIN {X 0,Y 418.491,Z 236.356,A -85,B 0,C 180,E1 -10253.247,E2 -10253.247} C_VEL
LIN {X 0,Y 418.339,Z 236.376,A -85,B 0,C 180,E1 -10255.18,E2 -10255.18} C_VEL
LIN {X 0,Y 418.541,Z 236.35,A -85,B 0,C 180,E1 -10258.074,E2 -10258.074} C_VEL
LIN {X 0,Y 418.67,Z 236.335,A -85,B 0,C 180,E1 -10259.998,E2 -10259.998} C_VEL
LIN {X 0,Y 418.506,Z 236.356,A -85,B 0,C 180,E1 -10262.886,E2 -10262.886} C_VEL
LIN {X 0,Y 418.488,Z 236.359,A -85,B 0,C 180,E1 -10266.749,E2 -10266.749} C_VEL
LIN {X 0,Y 418.392,Z 236.371,A -85,B 0,C 180,E1 -10268.693,E2 -10268.693} C_VEL
LIN {X 0,Y 418.213,Z 236.399,A -85,B 0,C 180,E1 -10271.632,E2 -10271.632} C_VEL
LIN {X 0,Y 418.124,Z 236.41,A -85,B 0,C 180,E1 -10272.871,E2 -10272.871} C_VEL
LIN {X 0,Y 417.983,Z 237.675,A -85,B 0,C 180,E1 -10274.607,E2 -10274.607} C_VEL
LIN {X 0,Y 417.883,Z 240.462,A -85,B 0,C 180,E1 -10277.619,E2 -10277.619} C_VEL
LIN {X 0,Y 417.76,Z 243.421,A -85,B 0,C 180,E1 -10280.686,E2 -10280.686} C_VEL
LIN {X 0,Y 417.651,Z 246.458,A -85,B 0,C 180,E1 -10283.817,E2 -10283.817} C_VEL
LIN {X 0,Y 417.55,Z 249.607,A -85,B 0,C 180,E1 -10287.027,E2 -10287.027} C_VEL
LIN {X 0,Y 417.503,Z 252.364,A -85,B 0,C 180,E1 -10289.807,E2 -10289.807} C_VEL
LIN {X 0,Y 421.016,Z 265.577,A -85,B 0,C 180,E1 -10290.434,E2 -10290.434} C_VEL
LIN {X 0,Y 422.505,Z 272.245,A -85,B 0,C 180,E1 -10290.816,E2 -10290.816} C_VEL
LIN {X 0,Y 422.029,Z 284.033,A -85,B 0,C 180,E1 -10291.502,E2 -10291.502} C_VEL
LIN {X 0,Y 421.315,Z 295.865,A -85,B 0,C 180,E1 -10292.401,E2 -10292.401} C_VEL
LIN {X 0,Y 420.581,Z 306.901,A -85,B 0,C 180,E1 -10293.463,E2 -10293.463} C_VEL
LIN {X 0,Y 419.846,Z 317.011,A -85,B 0,C 180,E1 -10294.688,E2 -10294.688} C_VEL
LIN {X 0,Y 419.249,Z 325.285,A -85,B 0,C 180,E1 -10295.922,E2 -10295.922} C_VEL
LIN {X 0,Y 418.691,Z 332.22,A -85,B 0,C 180,E1 -10297.175,E2 -10297.175} C_VEL
LIN {X 0,Y 418.247,Z 337.991,A -85,B 0,C 180,E1 -10298.44,E2 -10298.44} C_VEL
LIN {X 0,Y 417.881,Z 342.783,A -85,B 0,C 180,E1 -10299.721,E2 -10299.721} C_VEL
LIN {X 0,Y 417.634,Z 346.682,A -85,B 0,C 180,E1 -10301.015,E2 -10301.015} C_VEL
LIN {X 0,Y 417.423,Z 349.756,A -85,B 0,C 180,E1 -10302.332,E2 -10302.332} C_VEL
LIN {X 0,Y 417.221,Z 352.036,A -85,B 0,C 180,E1 -10303.677,E2 -10303.677} C_VEL
LIN {X 0,Y 417.105,Z 353.534,A -85,B 0,C 180,E1 -10305.043,E2 -10305.043} C_VEL
LIN {X 0,Y 417.042,Z 354.243,A -85,B 0,C 180,E1 -10306.435,E2 -10306.435} C_VEL
LIN {X 0,Y 417.022,Z 354.123,A -85,B 0,C 180,E1 -10307.858,E2 -10307.858} C_VEL
LIN {X 0,Y 417.114,Z 353.103,A -85,B 0,C 180,E1 -10309.303,E2 -10309.303} C_VEL
LIN {X 0,Y 417.243,Z 351.109,A -85,B 0,C 180,E1 -10310.785,E2 -10310.785} C_VEL
LIN {X 0,Y 417.502,Z 347.023,A -85,B 0,C 180,E1 -10312.7,E2 -10312.7} C_VEL
LIN {X 0,Y 417.826,Z 342.441,A -85,B 0,C 180,E1 -10314.233,E2 -10314.233} C_VEL
LIN {X 0,Y 418.212,Z 335.995,A -85,B 0,C 180,E1 -10315.892,E2 -10315.892} C_VEL
LIN {X 0,Y 418.735,Z 329.033,A -85,B 0,C 180,E1 -10317.298,E2 -10317.298} C_VEL
LIN {X 0,Y 419.344,Z 320.279,A -85,B 0,C 180,E1 -10318.726,E2 -10318.726} C_VEL
LIN {X 0,Y 420.037,Z 310.413,A -85,B 0,C 180,E1 -10320.024,E2 -10320.024} C_VEL
LIN {X 0,Y 420.762,Z 299.501,A -85,B 0,C 180,E1 -10321.165,E2 -10321.165} C_VEL
LIN {X 0,Y 421.444,Z 287.473,A -85,B 0,C 180,E1 -10322.166,E2 -10322.166} C_VEL
LIN {X 0,Y 422.063,Z 274.949,A -85,B 0,C 180,E1 -10322.955,E2 -10322.955} C_VEL
LIN {X 0,Y 422.141,Z 271.125,A -85,B 0,C 180,E1 -10323.159,E2 -10323.159} C_VEL
LIN {X 0,Y 419.239,Z 258.204,A -85,B 0,C 180,E1 -10323.827,E2 -10323.827} C_VEL
LIN {X 0,Y 417.432,Z 250.859,A -85,B 0,C 180,E1 -10324.141,E2 -10324.141} C_VEL
LIN {X 0,Y 417.434,Z 246.478,A -85,B 0,C 180,E1 -10328.261,E2 -10328.261} C_VEL
LIN {X 0,Y 417.509,Z 243.242,A -85,B 0,C 180,E1 -10331.348,E2 -10331.348} C_VEL
LIN {X 0,Y 417.58,Z 240.119,A -85,B 0,C 180,E1 -10334.379,E2 -10334.379} C_VEL
LIN {X 0,Y 417.719,Z 237.082,A -85,B 0,C 180,E1 -10337.367,E2 -10337.367} C_VEL
LIN {X 0,Y 417.771,Z 236.449,A -85,B 0,C 180,E1 -10338.354,E2 -10338.354} C_VEL
LIN {X 0,Y 418.176,Z 236.398,A -85,B 0,C 180,E1 -10341.301,E2 -10341.301} C_VEL
LIN {X 0,Y 418.444,Z 236.364,A -85,B 0,C 180,E1 -10343.249,E2 -10343.249} C_VEL
LIN {X 0,Y 418.329,Z 236.378,A -85,B 0,C 180,E1 -10345.182,E2 -10345.182} C_VEL
LIN {X 0,Y 418.529,Z 236.351,A -85,B 0,C 180,E1 -10348.076,E2 -10348.076} C_VEL
LIN {X 0,Y 418.65,Z 236.335,A -85,B 0,C 180,E1 -10350.037,E2 -10350.037} C_VEL
LIN {X 0,Y 417.83,Z 236.44,A -85,B 0,C 180,E1 -10350.84,E2 -10350.84} C_VEL
LIN {X 0,Y 414.806,Z 236.814,A -85,B 0,C 180,E1 -10352.141,E2 -10352.141} C_VEL
LIN {X 0,Y 412.339,Z 237.125,A -85,B 0,C 180,E1 -10353.193,E2 -10353.193} C_VEL
LIN {X 0,Y 411.314,Z 237.249,A -85,B 0,C 180,E1 -10354.007,E2 -10354.007} C_VEL
LIN {X 0,Y 411.244,Z 237.257,A -85,B 0,C 180,E1 -10354.283,E2 -10354.283} C_VEL
LIN {X 0,Y 411.445,Z 237.236,A -85,B 0,C 180,E1 -10356.868,E2 -10356.868} C_VEL
LIN {X 0,Y 411.293,Z 237.252,A -85,B 0,C 180,E1 -10359.839,E2 -10359.839} C_VEL
LIN {X 0,Y 411.298,Z 237.254,A -85,B 0,C 180,E1 -10363.11,E2 -10363.11} C_VEL
LIN {X 0,Y 411.242,Z 237.261,A -85,B 0,C 180,E1 -10366.89,E2 -10366.89} C_VEL
LIN {X 0,Y 411.241,Z 237.258,A -85,B 0,C 180,E1 -10369.987,E2 -10369.987} C_VEL
LIN {X 0,Y 411.21,Z 237.265,A -85,B 0,C 180,E1 -10373.148,E2 -10373.148} C_VEL
LIN {X 0,Y 411.226,Z 237.262,A -85,B 0,C 180,E1 -10376.382,E2 -10376.382} C_VEL
LIN {X 0,Y 411.187,Z 237.264,A -85,B 0,C 180,E1 -10379.714,E2 -10379.714} C_VEL
LIN {X 0,Y 411.194,Z 237.266,A -85,B 0,C 180,E1 -10383.157,E2 -10383.157} C_VEL
LIN {X 0,Y 411.185,Z 237.269,A -85,B 0,C 180,E1 -10386.555,E2 -10386.555} C_VEL
LIN {X 0,Y 411.218,Z 237.261,A -85,B 0,C 180,E1 -10389.732,E2 -10389.732} C_VEL
LIN {X 0,Y 411.215,Z 237.263,A -85,B 0,C 180,E1 -10393.129,E2 -10393.129} C_VEL
LIN {X 0,Y 411.231,Z 237.26,A -85,B 0,C 180,E1 -10395.872,E2 -10395.872} C_VEL
LIN {X 0,Y 411.205,Z 237.263,A -85,B 0,C 180,E1 -10399.502,E2 -10399.502} C_VEL
LIN {X 0,Y 411.198,Z 237.266,A -85,B 0,C 180,E1 -10402.029,E2 -10402.029} C_VEL
LIN {X 0,Y 411.2,Z 237.264,A -85,B 0,C 180,E1 -10405.668,E2 -10405.668} C_VEL
LIN {X 0,Y 411.195,Z 237.264,A -85,B 0,C 180,E1 -10409.155,E2 -10409.155} C_VEL
LIN {X 0,Y 411.256,Z 237.259,A -85,B 0,C 180,E1 -10412.524,E2 -10412.524} C_VEL
LIN {X 0,Y 411.224,Z 237.262,A -85,B 0,C 180,E1 -10415.787,E2 -10415.787} C_VEL
LIN {X 0,Y 411.194,Z 237.263,A -85,B 0,C 180,E1 -10418.968,E2 -10418.968} C_VEL
LIN {X 0,Y 411.251,Z 237.261,A -85,B 0,C 180,E1 -10422.087,E2 -10422.087} C_VEL
LIN {X 0,Y 411.259,Z 237.255,A -85,B 0,C 180,E1 -10425.149,E2 -10425.149} C_VEL
LIN {X 0,Y 411.283,Z 237.256,A -85,B 0,C 180,E1 -10428.169,E2 -10428.169} C_VEL
LIN {X 0,Y 411.439,Z 237.236,A -85,B 0,C 180,E1 -10432.193,E2 -10432.193} C_VEL
LIN {X 0,Y 411.471,Z 237.232,A -85,B 0,C 180,E1 -10434.12,E2 -10434.12} C_VEL
LIN {X 0,Y 411.513,Z 237.227,A -85,B 0,C 180,E1 -10438.044,E2 -10438.044} C_VEL
LIN {X 0,Y 411.643,Z 237.211,A -85,B 0,C 180,E1 -10440.002,E2 -10440.002} C_VEL
LIN {X 0,Y 411.459,Z 237.231,A -85,B 0,C 180,E1 -10442.939,E2 -10442.939} C_VEL
LIN {X 0,Y 411.427,Z 237.234,A -85,B 0,C 180,E1 -10446.869,E2 -10446.869} C_VEL
LIN {X 0,Y 411.295,Z 237.254,A -85,B 0,C 180,E1 -10449.84,E2 -10449.84} C_VEL
LIN {X 0,Y 411.31,Z 237.251,A -85,B 0,C 180,E1 -10453.105,E2 -10453.105} C_VEL
LIN {X 0,Y 411.263,Z 237.257,A -85,B 0,C 180,E1 -10456.89,E2 -10456.89} C_VEL
LIN {X 0,Y 411.236,Z 237.26,A -85,B 0,C 180,E1 -10459.988,E2 -10459.988} C_VEL
LIN {X 0,Y 411.207,Z 237.266,A -85,B 0,C 180,E1 -10463.149,E2 -10463.149} C_VEL
LIN {X 0,Y 411.239,Z 237.258,A -85,B 0,C 180,E1 -10466.382,E2 -10466.382} C_VEL
LIN {X 0,Y 411.207,Z 237.264,A -85,B 0,C 180,E1 -10469.714,E2 -10469.714} C_VEL
LIN {X 0,Y 411.213,Z 237.265,A -85,B 0,C 180,E1 -10473.157,E2 -10473.157} C_VEL
LIN {X 0,Y 411.199,Z 237.264,A -85,B 0,C 180,E1 -10476.553,E2 -10476.553} C_VEL
LIN {X 0,Y 411.216,Z 237.262,A -85,B 0,C 180,E1 -10479.728,E2 -10479.728} C_VEL
LIN {X 0,Y 411.18,Z 237.265,A -85,B 0,C 180,E1 -10483.134,E2 -10483.134} C_VEL
LIN {X 0,Y 411.179,Z 237.277,A -85,B 0,C 180,E1 -10486.396,E2 -10486.396} C_VEL
LIN {X 0,Y 412.343,Z 243.292,A -85,B 0,C 180,E1 -10489.633,E2 -10489.633} C_VEL
LIN {X 0,Y 413.228,Z 248.458,A -85,B 0,C 180,E1 -10492.246,E2 -10492.246} C_VEL
LIN {X 0,Y 413.528,Z 252.304,A -85,B 0,C 180,E1 -10494.103,E2 -10494.103} C_VEL
LIN {X 0,Y 413.002,Z 258.756,A -85,B 0,C 180,E1 -10497.006,E2 -10497.006} C_VEL
LIN {X 0,Y 412.458,Z 265.207,A -85,B 0,C 180,E1 -10499.824,E2 -10499.824} C_VEL
LIN {X 0,Y 412.025,Z 271.725,A -85,B 0,C 180,E1 -10502.577,E2 -10502.577} C_VEL
LIN {X 0,Y 411.533,Z 279.56,A -85,B 0,C 180,E1 -10505.803,E2 -10505.803} C_VEL
LIN {X 0,Y 411.121,Z 287.418,A -85,B 0,C 180,E1 -10508.961,E2 -10508.961} C_VEL
LIN {X 0,Y 410.723,Z 296.13,A -85,B 0,C 180,E1 -10512.398,E2 -10512.398} C_VEL
LIN {X 0,Y 413.1,Z 310.786,A -85,B 0,C 180,E1 -10512.96,E2 -10512.96} C_VEL
LIN {X 0,Y 414.851,Z 323.576,A -85,B 0,C 180,E1 -10513.641,E2 -10513.641} C_VEL
LIN {X 0,Y 414.263,Z 335.298,A -85,B 0,C 180,E1 -10514.376,E2 -10514.376} C_VEL
LIN {X 0,Y 413.542,Z 346.012,A -85,B 0,C 180,E1 -10515.231,E2 -10515.231} C_VEL
LIN {X 0,Y 412.873,Z 355.909,A -85,B 0,C 180,E1 -10516.213,E2 -10516.213} C_VEL
LIN {X 0,Y 412.148,Z 365.934,A -85,B 0,C 180,E1 -10517.442,E2 -10517.442} C_VEL
LIN {X 0,Y 411.35,Z 375.655,A -85,B 0,C 180,E1 -10518.918,E2 -10518.918} C_VEL
LIN {X 0,Y 410.829,Z 383.42,A -85,B 0,C 180,E1 -10520.398,E2 -10520.398} C_VEL
LIN {X 0,Y 410.358,Z 390.567,A -85,B 0,C 180,E1 -10522.125,E2 -10522.125} C_VEL
